C09152=1150.705,51.432,-50.728,-179.726,6.322,149.066
C09153=1150.710,51.184,-50.712,-179.728,6.321,149.066
C09154=1150.715,50.934,-50.696,-179.731,6.319,149.067
C09155=1150.720,50.684,-50.680,-179.733,6.319,149.067
C09156=1150.725,50.435,-50.665,-179.736,6.317,149.068
C09157=1150.730,50.186,-50.650,-179.739,6.317,149.069
C09158=1150.736,49.936,-50.634,-179.741,6.316,149.069
C09159=1150.740,49.686,-50.618,-179.744,6.314,149.069
C09160=1150.745,49.437,-50.603,-179.746,6.314,149.070
C09161=1150.750,49.188,-50.588,-179.749,6.312,149.071
C09162=1150.755,48.938,-50.571,-179.752,6.311,149.071
C09163=1150.760,48.689,-50.555,-179.754,6.310,149.072
C09164=1150.765,48.440,-50.540,-179.757,6.309,149.072
C09165=1150.770,48.190,-50.525,-179.760,6.308,149.073
C09166=1150.775,47.940,-50.509,-179.762,6.307,149.073
C09167=1150.780,47.691,-50.494,-179.765,6.306,149.074
C09168=1150.785,47.442,-50.478,-179.767,6.305,149.074
C09169=1150.791,47.192,-50.463,-179.770,6.304,149.075
C09170=1150.795,46.942,-50.447,-179.773,6.303,149.075
C09171=1150.800,46.693,-50.432,-179.775,6.302,149.076
C09172=1150.805,46.444,-50.416,-179.778,6.301,149.077
C09173=1150.811,46.194,-50.401,-179.780,6.300,149.077
C09174=1150.815,45.945,-50.386,-179.784,6.298,149.078
C09175=1150.820,45.695,-50.370,-179.786,6.298,149.078
C09176=1150.825,45.446,-50.355,-179.789,6.296,149.079
C09177=1150.830,45.197,-50.339,-179.791,6.295,149.079
C09178=1150.836,44.947,-50.324,-179.793,6.295,149.080
C09179=1150.841,44.697,-50.309,-179.797,6.293,149.080
C09180=1150.845,44.447,-50.293,-179.799,6.292,149.081
C09181=1150.851,44.198,-50.278,-179.801,6.291,149.081
C09182=1150.855,43.949,-50.263,-179.804,6.290,149.082
C09183=1150.861,43.699,-50.247,-179.807,6.289,149.082
C09184=1150.865,43.450,-50.232,-179.810,6.288,149.083
C09185=1150.870,43.200,-50.216,-179.812,6.287,149.084
C09186=1150.876,42.951,-50.201,-179.815,6.286,149.084
C09187=1150.881,42.701,-50.186,-179.817,6.285,149.085
C09188=1150.886,42.452,-50.171,-179.820,6.284,149.085
C09189=1150.891,42.203,-50.156,-179.822,6.283,149.086
C09190=1150.896,41.953,-50.140,-179.825,6.282,149.086
C09191=1150.901,41.704,-50.125,-179.828,6.281,149.087
C09192=1150.906,41.453,-50.110,-179.830,6.280,149.087
C09193=1150.910,41.204,-50.095,-179.833,6.279,149.088
C09194=1150.916,40.955,-50.079,-179.835,6.278,149.088
C09195=1150.920,40.706,-50.064,-179.838,6.277,149.089
C09196=1150.926,40.456,-50.049,-179.841,6.276,149.090
C09197=1150.932,40.206,-50.034,-179.843,6.275,149.090
C09198=1150.936,39.957,-50.019,-179.846,6.274,149.091
C09199=1150.942,39.708,-50.003,-179.848,6.273,149.091
C09200=1150.946,39.458,-49.989,-179.851,6.272,149.092
C09201=1150.951,39.208,-49.973,-179.854,6.271,149.092
C09202=1150.956,38.959,-49.958,-179.856,6.270,149.093
C09203=1150.961,38.709,-49.944,-179.859,6.269,149.093
C09204=1150.966,38.460,-49.928,-179.861,6.268,149.094
C09205=1150.971,38.211,-49.913,-179.864,6.267,149.094
C09206=1150.976,37.961,-49.898,-179.867,6.266,149.095
C09207=1150.981,37.712,-49.883,-179.869,6.265,149.095
C09208=1150.987,37.462,-49.868,-179.872,6.264,149.096
C09209=1150.992,37.213,-49.853,-179.874,6.263,149.097
C09210=1150.997,36.963,-49.838,-179.877,6.262,149.097
C09211=1151.002,36.714,-49.823,-179.880,6.261,149.098
C09212=1151.007,36.464,-49.809,-179.882,6.260,149.098
C09213=1151.012,36.215,-49.793,-179.884,6.259,149.099
C09214=1151.017,35.965,-49.779,-179.888,6.258,149.099
C09215=1151.022,35.716,-49.763,-179.890,6.257,149.100
C09216=1151.026,35.466,-49.748,-179.893,6.256,149.100
C09217=1151.031,35.216,-49.734,-179.895,6.255,149.101
C09218=1151.037,34.967,-49.718,-179.897,6.254,149.101
C09219=1151.042,34.717,-49.704,-179.901,6.253,149.102
C09220=1151.047,34.468,-49.688,-179.903,6.252,149.103
C09221=1151.052,34.218,-49.674,-179.906,6.252,149.103
C09222=1151.057,33.969,-49.659,-179.908,6.250,149.104
C09223=1151.062,33.719,-49.644,-179.910,6.249,149.104
C09224=1151.067,33.470,-49.629,-179.913,6.249,149.105
C09225=1151.072,33.220,-49.615,-179.916,6.247,149.105
C09226=1151.077,32.971,-49.599,-179.918,6.247,149.106
C09227=1151.082,32.721,-49.585,-179.921,6.246,149.106
C09228=1151.087,32.472,-49.570,-179.924,6.245,149.107
C09229=1151.093,32.222,-49.555,-179.926,6.244,149.108
C09230=1151.097,31.973,-49.540,-179.929,6.243,149.108
C09231=1151.102,31.723,-49.526,-179.931,6.242,149.109
C09232=1151.108,31.474,-49.512,-179.934,6.241,149.109
C09233=1151.113,31.225,-49.496,-179.937,6.240,149.110
C09234=1151.118,30.975,-49.482,-179.939,6.239,149.110
C09235=1151.123,30.726,-49.467,-179.942,6.238,149.111
C09236=1151.128,30.476,-49.453,-179.944,6.237,149.111
C09237=1151.133,30.226,-49.438,-179.947,6.236,149.112
C09238=1151.138,29.977,-49.423,-179.949,6.235,149.113
C09239=1151.143,29.727,-49.408,-179.952,6.234,149.113
C09240=1151.148,29.478,-49.394,-179.955,6.233,149.114
C09241=1151.153,29.228,-49.379,-179.957,6.232,149.114
C09242=1151.158,28.979,-49.364,-179.959,6.232,149.115
C09243=1151.163,28.729,-49.350,-179.962,6.230,149.115
C09244=1151.168,28.480,-49.335,-179.965,6.230,149.116
C09245=1151.173,28.230,-49.321,-179.967,6.229,149.116
C09246=1151.179,27.961,-49.304,-179.970,6.228,149.117
C09247=1151.185,27.693,-49.289,-179.973,6.227,149.118
C09248=1151.190,27.424,-49.274,-179.976,6.226,149.118
C09249=1151.196,27.154,-49.258,-179.978,6.225,149.119
C09250=1151.201,26.905,-49.244,-179.981,6.224,149.119
C09251=1151.205,26.656,-49.229,-179.984,6.223,149.120
C09252=1151.210,26.406,-49.214,-179.986,6.222,149.120
C09253=1151.215,26.156,-49.200,-179.989,6.221,149.121
C09254=1151.220,25.907,-49.186,-179.991,6.220,149.122
C09255=1151.225,25.657,-49.171,-179.994,6.220,149.122
C09256=1151.231,25.408,-49.156,-179.997,6.218,149.123
C09257=1151.236,25.158,-49.142,-179.999,6.217,149.123
C09258=1151.241,24.909,-49.128,179.998,6.217,149.124
C09259=1151.246,24.659,-49.113,179.996,6.216,149.124
C09260=1151.251,24.409,-49.099,179.993,6.215,149.125
C09261=1151.256,24.160,-49.084,179.991,6.214,149.125
C09262=1151.261,23.911,-49.070,179.988,6.213,149.126
C09263=1151.266,23.661,-49.056,179.985,6.212,149.127
C09264=1151.271,23.412,-49.042,179.983,6.211,149.127
C09265=1151.276,23.162,-49.027,179.981,6.211,149.128
C09266=1151.282,22.912,-49.013,179.978,6.210,149.128
C09267=1151.287,22.662,-48.998,179.975,6.208,149.129
C09268=1151.292,22.413,-48.984,179.973,6.208,149.129
C09269=1151.297,22.164,-48.969,179.970,6.207,149.130
C09270=1151.302,21.914,-48.955,179.968,6.206,149.130
C09271=1151.307,21.665,-48.941,179.965,6.205,149.131
C09272=1151.312,21.415,-48.926,179.963,6.204,149.132
C09273=1151.317,21.166,-48.913,179.960,6.204,149.132
C09274=1151.322,20.916,-48.898,179.957,6.202,149.133
C09275=1151.327,20.667,-48.884,179.955,6.202,149.133
C09276=1151.332,20.417,-48.870,179.953,6.201,149.134
C09277=1151.337,20.167,-48.855,179.949,6.200,149.135
C09278=1151.343,19.918,-48.842,179.947,6.199,149.135
C09279=1151.348,19.668,-48.827,179.945,6.198,149.136
C09280=1151.353,19.419,-48.813,179.942,6.198,149.136
C09281=1151.358,19.169,-48.799,179.940,6.196,149.137
C09282=1151.363,18.920,-48.785,179.937,6.195,149.137
C09283=1151.368,18.670,-48.771,179.935,6.195,149.138
C09284=1151.373,18.421,-48.756,179.932,6.194,149.138
C09285=1151.378,18.171,-48.742,179.929,6.193,149.139
C09286=1151.384,17.922,-48.728,179.927,6.192,149.140
C09287=1151.388,17.673,-48.714,179.925,6.191,149.140
C09288=1151.393,17.422,-48.701,179.922,6.191,149.141
C09289=1151.398,17.172,-48.687,179.919,6.189,149.141
C09290=1151.404,16.923,-48.673,179.917,6.189,149.142
C09291=1151.409,16.674,-48.658,179.914,6.188,149.142
C09292=1151.414,16.424,-48.644,179.912,6.187,149.143
C09293=1151.419,16.175,-48.630,179.909,6.186,149.143
C09294=1151.424,15.925,-48.616,179.906,6.185,149.144
C09295=1151.429,15.676,-48.602,179.904,6.185,149.145
C09296=1151.434,15.425,-48.588,179.902,6.184,149.145
C09297=1151.439,15.177,-48.575,179.899,6.182,149.146
C09298=1151.444,14.927,-48.560,179.897,6.182,149.146
C09299=1151.449,14.677,-48.546,179.894,6.181,149.147
C09300=1151.455,14.428,-48.532,179.892,6.180,149.147
C09301=1151.459,14.178,-48.518,179.889,6.180,149.148
C09302=1151.465,13.928,-48.504,179.886,6.178,149.148
C09303=1151.470,13.679,-48.491,179.884,6.178,149.149
C09304=1151.475,13.430,-48.477,179.881,6.177,149.150
C09305=1151.479,13.180,-48.463,179.879,6.177,149.150
C09306=1151.485,12.930,-48.449,179.876,6.175,149.151
C09307=1151.490,12.681,-48.435,179.873,6.174,149.151
C09308=1151.495,12.431,-48.421,179.871,6.174,149.152
C09309=1151.500,12.182,-48.408,179.869,6.173,149.153
C09310=1151.505,11.932,-48.394,179.866,6.172,149.153
C09311=1151.511,11.683,-48.380,179.864,6.171,149.153
C09312=1151.516,11.433,-48.366,179.861,6.170,149.154
C09313=1151.521,11.183,-48.352,179.859,6.169,149.155
C09314=1151.526,10.934,-48.339,179.856,6.169,149.155
C09315=1151.531,10.684,-48.325,179.854,6.168,149.156
C09316=1151.536,10.434,-48.311,179.851,6.167,149.156
C09317=1151.542,10.185,-48.297,179.849,6.166,149.157
C09318=1151.546,9.936,-48.283,179.846,6.166,149.158
C09319=1151.552,9.686,-48.270,179.844,6.165,149.158
C09320=1151.557,9.436,-48.256,179.841,6.164,149.159
C09321=1151.561,9.187,-48.242,179.838,6.163,149.159
C09322=1151.567,8.937,-48.229,179.836,6.162,149.160
C09323=1151.572,8.688,-48.215,179.834,6.162,149.160
C09324=1151.577,8.439,-48.201,179.831,6.161,149.161
C09325=1151.582,8.189,-48.188,179.829,6.160,149.161
C09326=1151.587,7.940,-48.174,179.825,6.159,149.162
C09327=1151.593,7.689,-48.160,179.823,6.158,149.163
C09328=1151.597,7.440,-48.147,179.821,6.158,149.163
C09329=1151.603,7.190,-48.134,179.818,6.157,149.164
C09330=1151.608,6.941,-48.119,179.816,6.156,149.164
C09331=1151.613,6.691,-48.107,179.813,6.155,149.165
C09332=1151.618,6.442,-48.092,179.811,6.154,149.165
C09333=1151.623,6.193,-48.079,179.808,6.154,149.166
C09334=1151.628,5.942,-48.066,179.806,6.153,149.167
C09335=1151.633,5.693,-48.052,179.803,6.152,149.167
C09336=1151.639,5.443,-48.038,179.801,6.152,149.168
C09337=1151.643,5.194,-48.024,179.798,6.150,149.168
C09338=1151.649,4.944,-48.011,179.796,6.149,149.169
C09339=1151.653,4.694,-47.998,179.793,6.149,149.170
C09340=1151.659,4.445,-47.984,179.791,6.148,149.170
C09341=1151.664,4.195,-47.971,179.788,6.148,149.171
C09342=1151.669,3.946,-47.957,179.786,6.147,149.171
C09343=1151.674,3.696,-47.944,179.783,6.146,149.172
C09344=1151.679,3.447,-47.931,179.781,6.145,149.172
C09345=1151.684,3.197,-47.917,179.778,6.144,149.173
C09346=1151.690,2.947,-47.904,179.776,6.144,149.173
C09347=1151.694,2.698,-47.890,179.773,6.143,149.174
C09348=1151.700,2.448,-47.877,179.771,6.142,149.175
C09349=1151.704,2.199,-47.863,179.768,6.141,149.175
C09350=1151.711,1.929,-47.849,179.766,6.140,149.176
C09351=1151.716,1.660,-47.834,179.763,6.140,149.176
C09352=1151.721,1.390,-47.821,179.760,6.139,149.177
C09353=1151.727,1.121,-47.806,179.758,6.138,149.178
C09354=1151.732,0.871,-47.792,179.755,6.137,149.178
C09355=1151.737,0.622,-47.779,179.753,6.137,149.179
C09356=1151.743,0.372,-47.766,179.750,6.136,149.179
C09357=1151.748,0.123,-47.753,179.748,6.135,149.180
C09358=1151.753,-0.127,-47.739,179.745,6.134,149.181
C09359=1151.758,-0.376,-47.726,179.742,6.133,149.181
C09360=1151.763,-0.627,-47.713,179.740,6.133,149.182
C09361=1151.768,-0.876,-47.700,179.738,6.132,149.182
C09362=1151.774,-1.125,-47.686,179.735,6.132,149.183
C09363=1151.778,-1.375,-47.673,179.733,6.131,149.183
C09364=1151.784,-1.625,-47.660,179.731,6.130,149.184
C09365=1151.789,-1.875,-47.647,179.728,6.130,149.184
C09366=1151.793,-2.123,-47.634,179.725,6.128,149.185
C09367=1151.799,-2.373,-47.620,179.723,6.127,149.186
C09368=1151.804,-2.623,-47.607,179.720,6.127,149.186
C09369=1151.810,-2.873,-47.594,179.718,6.126,149.187
C09370=1151.814,-3.123,-47.581,179.716,6.125,149.187
C09371=1151.820,-3.372,-47.567,179.713,6.125,149.188
C09372=1151.825,-3.621,-47.555,179.711,6.124,149.188
C09373=1151.829,-3.871,-47.542,179.708,6.124,149.189
C09374=1151.835,-4.121,-47.529,179.705,6.122,149.190
C09375=1151.840,-4.371,-47.516,179.703,6.122,149.190
C09376=1151.845,-4.620,-47.502,179.700,6.121,149.191
C09377=1151.850,-4.869,-47.489,179.698,6.120,149.191
C09378=1151.855,-5.119,-47.476,179.696,6.120,149.192
C09379=1151.861,-5.369,-47.463,179.693,6.119,149.193
C09380=1151.866,-5.618,-47.450,179.691,6.118,149.193
C09381=1151.870,-5.868,-47.437,179.688,6.118,149.194
C09382=1151.876,-6.117,-47.424,179.686,6.117,149.194
C09383=1151.881,-6.367,-47.412,179.683,6.116,149.195
C09384=1151.887,-6.617,-47.398,179.680,6.115,149.195
C09385=1151.892,-6.866,-47.385,179.678,6.115,149.196
C09386=1151.897,-7.115,-47.372,179.676,6.114,149.197
C09387=1151.902,-7.365,-47.359,179.673,6.113,149.197
C09388=1151.907,-7.615,-47.346,179.671,6.113,149.198
C09389=1151.912,-7.864,-47.333,179.669,6.112,149.198
C09390=1151.917,-8.114,-47.320,179.666,6.111,149.199
C09391=1151.923,-8.364,-47.307,179.664,6.110,149.199
C09392=1151.928,-8.613,-47.295,179.661,6.110,149.200
C09393=1151.932,-8.863,-47.282,179.659,6.109,149.200
C09394=1151.938,-9.113,-47.268,179.656,6.108,149.201
C09395=1151.943,-9.362,-47.256,179.654,6.107,149.202
C09396=1151.948,-9.612,-47.243,179.651,6.107,149.202
C09397=1151.953,-9.861,-47.230,179.649,6.106,149.203
C09398=1151.959,-10.111,-47.217,179.646,6.106,149.203
C09399=1151.964,-10.360,-47.204,179.644,6.105,149.204
C09400=1151.968,-10.610,-47.192,179.641,6.104,149.205
C09401=1151.973,-10.860,-47.179,179.639,6.103,149.205
C09402=1151.979,-11.109,-47.166,179.636,6.103,149.206
C09403=1151.984,-11.360,-47.153,179.634,6.102,149.206
C09404=1151.989,-11.609,-47.141,179.632,6.102,149.207
C09405=1151.994,-11.859,-47.128,179.629,6.101,149.207
C09406=1152.000,-12.108,-47.116,179.627,6.101,149.208
C09407=1152.005,-12.358,-47.102,179.624,6.099,149.209
C09408=1152.010,-12.608,-47.089,179.621,6.099,149.209
C09409=1152.015,-12.857,-47.077,179.619,6.098,149.210
C09410=1152.020,-13.106,-47.064,179.616,6.097,149.210
C09411=1152.025,-13.356,-47.051,179.614,6.097,149.211
C09412=1152.031,-13.606,-47.039,179.612,6.096,149.211
C09413=1152.036,-13.856,-47.026,179.609,6.095,149.212
C09414=1152.041,-14.105,-47.014,179.607,6.094,149.213
C09415=1152.046,-14.354,-47.001,179.605,6.094,149.213
C09416=1152.051,-14.604,-46.988,179.602,6.093,149.214
C09417=1152.056,-14.854,-46.975,179.600,6.093,149.214
C09418=1152.061,-15.104,-46.964,179.598,6.092,149.215
C09419=1152.067,-15.353,-46.950,179.595,6.092,149.216
C09420=1152.072,-15.603,-46.938,179.593,6.091,149.216
C09421=1152.077,-15.853,-46.925,179.590,6.090,149.217
C09422=1152.082,-16.103,-46.913,179.588,6.090,149.217
C09423=1152.087,-16.352,-46.900,179.585,6.089,149.218
C09424=1152.092,-16.601,-46.888,179.583,6.088,149.218
C09425=1152.098,-16.851,-46.875,179.580,6.088,149.219
C09426=1152.102,-17.101,-46.863,179.578,6.087,149.219
C09427=1152.108,-17.350,-46.850,179.575,6.086,149.220
C09428=1152.113,-17.600,-46.837,179.573,6.085,149.221
C09429=1152.119,-17.849,-46.824,179.570,6.085,149.221
C09430=1152.124,-18.099,-46.813,179.568,6.084,149.222
C09431=1152.129,-18.349,-46.800,179.565,6.083,149.223
C09432=1152.134,-18.598,-46.787,179.563,6.083,149.223
C09433=1152.139,-18.849,-46.775,179.560,6.082,149.224
C09434=1152.144,-19.098,-46.763,179.558,6.081,149.224
C09435=1152.149,-19.347,-46.750,179.556,6.081,149.225
C09436=1152.155,-19.597,-46.738,179.553,6.080,149.225
C09437=1152.160,-19.847,-46.725,179.551,6.079,149.226
C09438=1152.165,-20.096,-46.713,179.549,6.079,149.226
C09439=1152.170,-20.346,-46.701,179.546,6.078,149.227
C09440=1152.176,-20.595,-46.688,179.544,6.078,149.228
C09441=1152.180,-20.845,-46.675,179.542,6.077,149.228
C09442=1152.185,-21.095,-46.664,179.539,6.076,149.229
C09443=1152.191,-21.344,-46.651,179.537,6.076,149.229
C09444=1152.196,-21.594,-46.639,179.534,6.075,149.230
C09445=1152.201,-21.844,-46.626,179.532,6.074,149.230
C09446=1152.207,-22.094,-46.615,179.529,6.074,149.231
C09447=1152.212,-22.343,-46.602,179.527,6.073,149.232
C09448=1152.217,-22.592,-46.589,179.524,6.073,149.232
C09449=1152.222,-22.842,-46.577,179.522,6.072,149.233
C09450=1152.227,-23.091,-46.565,179.520,6.072,149.233
C09451=1152.233,-23.341,-46.553,179.517,6.071,149.234
C09452=1152.237,-23.591,-46.540,179.515,6.070,149.235
C09453=1152.243,-23.841,-46.528,179.512,6.070,149.235
C09454=1152.248,-24.110,-46.515,179.510,6.069,149.236
C09455=1152.254,-24.381,-46.502,179.508,6.068,149.236
C09456=1152.260,-24.651,-46.488,179.505,6.068,149.237
C09457=1152.265,-24.920,-46.475,179.502,6.067,149.238
C09458=1152.271,-25.170,-46.463,179.500,6.066,149.238
C09459=1152.276,-25.420,-46.451,179.497,6.065,149.239
C09460=1152.281,-25.670,-46.439,179.495,6.065,149.239
C09461=1152.286,-25.919,-46.427,179.493,6.065,149.240
C09462=1152.291,-26.169,-46.415,179.490,6.064,149.240
C09463=1152.297,-26.418,-46.403,179.488,6.063,149.241
C09464=1152.302,-26.668,-46.390,179.486,6.063,149.242
C09465=1152.307,-26.918,-46.378,179.483,6.062,149.242
C09466=1152.312,-27.168,-46.365,179.481,6.062,149.243
C09467=1152.317,-27.418,-46.353,179.479,6.061,149.243
C09468=1152.322,-27.668,-46.342,179.476,6.061,149.244
C09469=1152.327,-27.917,-46.330,179.474,6.060,149.244
C09470=1152.332,-28.167,-46.318,179.471,6.059,149.245
C09471=1152.338,-28.417,-46.306,179.469,6.059,149.246
C09472=1152.343,-28.666,-46.293,179.466,6.058,149.246
C09473=1152.348,-28.916,-46.281,179.464,6.057,149.247
C09474=1152.353,-29.165,-46.269,179.461,6.057,149.247
C09475=1152.358,-29.415,-46.257,179.459,6.056,149.248
C09476=1152.364,-29.665,-46.246,179.457,6.056,149.249
C09477=1152.369,-29.913,-46.233,179.454,6.055,149.249
C09478=1152.375,-30.163,-46.221,179.452,6.054,149.250
C09479=1152.379,-30.413,-46.210,179.450,6.054,149.250
C09480=1152.385,-30.663,-46.198,179.447,6.053,149.251
C09481=1152.390,-30.912,-46.186,179.445,6.052,149.251
C09482=1152.395,-31.162,-46.174,179.442,6.052,149.252
C09483=1152.401,-31.412,-46.162,179.440,6.051,149.253
C09484=1152.405,-31.661,-46.150,179.438,6.050,149.253
C09485=1152.411,-31.911,-46.138,179.435,6.050,149.254
C09486=1152.416,-32.161,-46.126,179.433,6.049,149.254
C09487=1152.421,-32.411,-46.114,179.430,6.049,149.255
C09488=1152.426,-32.660,-46.102,179.428,6.048,149.255
C09489=1152.431,-32.910,-46.090,179.425,6.048,149.256
C09490=1152.437,-33.160,-46.078,179.424,6.048,149.257
C09491=1152.442,-33.410,-46.067,179.421,6.047,149.257
C09492=1152.447,-33.659,-46.055,179.419,6.046,149.258
C09493=1152.452,-33.909,-46.043,179.417,6.046,149.258
C09494=1152.457,-34.158,-46.031,179.414,6.045,149.259
C09495=1152.463,-34.407,-46.020,179.412,6.044,149.259
C09496=1152.468,-34.657,-46.008,179.409,6.044,149.260
C09497=1152.474,-34.907,-45.996,179.407,6.043,149.261
C09498=1152.478,-35.156,-45.984,179.404,6.043,149.261
C09499=1152.483,-35.406,-45.972,179.402,6.042,149.262
C09500=1152.489,-35.656,-45.960,179.399,6.042,149.263
C09501=1152.493,-35.906,-45.949,179.397,6.041,149.263
C09502=1152.499,-36.156,-45.937,179.395,6.040,149.264
C09503=1152.504,-36.406,-45.925,179.392,6.040,149.264
C09504=1152.510,-36.655,-45.914,179.390,6.039,149.265
C09505=1152.515,-36.904,-45.902,179.388,6.039,149.265
C09506=1152.520,-37.154,-45.890,179.386,6.038,149.266
C09507=1152.525,-37.403,-45.879,179.383,6.038,149.267
C09508=1152.530,-37.653,-45.867,179.381,6.037,149.267
C09509=1152.536,-37.903,-45.855,179.378,6.037,149.268
C09510=1152.540,-38.153,-45.844,179.376,6.036,149.268
C09511=1152.546,-38.402,-45.832,179.374,6.036,149.269
C09512=1152.552,-38.652,-45.820,179.371,6.035,149.269
C09513=1152.557,-38.902,-45.809,179.369,6.034,149.270
C09514=1152.562,-39.152,-45.797,179.367,6.034,149.271
C09515=1152.567,-39.401,-45.786,179.364,6.033,149.271
C09516=1152.572,-39.651,-45.774,179.362,6.032,149.272
C09517=1152.578,-39.900,-45.762,179.360,6.032,149.272
C09518=1152.583,-40.150,-45.751,179.357,6.032,149.273
C09519=1152.588,-40.400,-45.739,179.355,6.031,149.273
C09520=1152.593,-40.650,-45.728,179.353,6.031,149.274
C09521=1152.598,-40.900,-45.716,179.350,6.030,149.275
C09522=1152.604,-41.149,-45.705,179.348,6.030,149.275
C09523=1152.609,-41.398,-45.693,179.346,6.029,149.276
C09524=1152.614,-41.648,-45.682,179.343,6.028,149.276
C09525=1152.619,-41.898,-45.670,179.341,6.028,149.277
C09526=1152.624,-42.148,-45.659,179.339,6.027,149.277
C09527=1152.630,-42.397,-45.647,179.337,6.027,149.278
C09528=1152.635,-42.647,-45.635,179.334,6.026,149.279
C09529=1152.640,-42.896,-45.624,179.332,6.026,149.279
C09530=1152.646,-43.147,-45.613,179.329,6.025,149.280
C09531=1152.650,-43.397,-45.601,179.327,6.025,149.280
C09532=1152.657,-43.646,-45.590,179.325,6.024,149.281
C09533=1152.661,-43.895,-45.579,179.322,6.024,149.282
C09534=1152.667,-44.145,-45.567,179.320,6.023,149.282
C09535=1152.671,-44.395,-45.555,179.317,6.022,149.283
C09536=1152.677,-44.644,-45.545,179.316,6.022,149.283
C09537=1152.682,-44.894,-45.533,179.313,6.022,149.284
C09538=1152.687,-45.144,-45.522,179.311,6.021,149.284
C09539=1152.692,-45.394,-45.510,179.308,6.020,149.285
C09540=1152.698,-45.643,-45.499,179.306,6.020,149.286
C09541=1152.703,-45.893,-45.487,179.304,6.019,149.286
C09542=1152.708,-46.143,-45.476,179.301,6.019,149.287
C09543=1152.713,-46.393,-45.464,179.299,6.018,149.287
C09544=1152.719,-46.642,-45.454,179.297,6.018,149.288
C09545=1152.724,-46.892,-45.442,179.295,6.018,149.288
C09546=1152.729,-47.142,-45.431,179.292,6.017,149.289
C09547=1152.734,-47.391,-45.420,179.290,6.016,149.290
C09548=1152.740,-47.640,-45.408,179.287,6.016,149.290
C09549=1152.745,-47.891,-45.397,179.285,6.015,149.291
C09550=1152.750,-48.141,-45.386,179.283,6.014,149.291
C09551=1152.755,-48.390,-45.375,179.281,6.015,149.292
C09552=1152.760,-48.639,-45.363,179.278,6.014,149.292
C09553=1152.766,-48.890,-45.352,179.276,6.013,149.293
C09554=1152.771,-49.139,-45.341,179.274,6.013,149.294
C09555=1152.777,-49.389,-45.329,179.271,6.012,149.294
C09556=1152.782,-49.639,-45.319,179.269,6.012,149.295
C09557=1152.787,-49.888,-45.308,179.266,6.011,149.295
C09558=1152.793,-50.159,-45.296,179.264,6.010,149.296
C09559=1152.798,-50.430,-45.283,179.262,6.010,149.296
C09560=1152.804,-50.700,-45.271,179.259,6.009,149.297
C09561=1152.810,-50.970,-45.259,179.256,6.009,149.298
C09562=1152.815,-51.220,-45.248,179.255,6.009,149.298
C09563=1152.820,-51.470,-45.237,179.252,6.008,149.299
C09564=1152.825,-51.719,-45.225,179.250,6.008,149.300
C09565=1152.831,-51.969,-45.215,179.248,6.007,149.300
C09566=1152.836,-52.219,-45.204,179.245,6.006,149.301
C09567=1152.841,-52.469,-45.193,179.243,6.006,149.301
C09568=1152.847,-52.718,-45.182,179.240,6.005,149.302
C09569=1152.851,-52.968,-45.170,179.239,6.005,149.302
C09570=1152.856,-53.218,-45.160,179.236,6.005,149.303
C09571=1152.862,-53.467,-45.148,179.234,6.004,149.304
C09572=1152.867,-53.717,-45.138,179.231,6.003,149.304
C09573=1152.872,-53.967,-45.126,179.229,6.003,149.305
C09574=1152.877,-54.216,-45.115,179.227,6.002,149.305
C09575=1152.883,-54.467,-45.104,179.225,6.003,149.306
C09576=1152.888,-54.716,-45.093,179.222,6.002,149.306
C09577=1152.893,-54.966,-45.083,179.220,6.001,149.307
C09578=1152.898,-55.215,-45.071,179.218,6.001,149.308
C09579=1152.904,-55.465,-45.061,179.215,6.000,149.308
C09580=1152.909,-55.715,-45.049,179.213,6.000,149.309
C09581=1152.915,-55.964,-45.039,179.211,5.999,149.309
C09582=1152.919,-56.214,-45.028,179.208,5.999,149.310
C09583=1152.924,-56.464,-45.017,179.206,5.998,149.310
C09584=1152.930,-56.714,-45.006,179.204,5.998,149.311
C09585=1152.935,-56.964,-44.995,179.201,5.997,149.312
C09586=1152.941,-57.213,-44.984,179.200,5.997,149.312
C09587=1152.946,-57.463,-44.974,179.197,5.997,149.313
C09588=1152.951,-57.712,-44.963,179.195,5.996,149.313
C09589=1152.957,-57.962,-44.952,179.192,5.995,149.314
C09590=1152.962,-58.212,-44.940,179.190,5.995,149.314
C09591=1152.967,-58.462,-44.930,179.188,5.995,149.315
C09592=1152.972,-58.711,-44.919,179.186,5.994,149.316
C09593=1152.977,-58.961,-44.909,179.184,5.994,149.316
C09594=1152.982,-59.210,-44.897,179.181,5.993,149.317
C09595=1152.988,-59.460,-44.886,179.179,5.992,149.317
C09596=1152.993,-59.710,-44.876,179.177,5.992,149.318
C09597=1152.999,-59.959,-44.865,179.174,5.992,149.318
C09598=1153.004,-60.210,-44.854,179.172,5.991,149.319
C09599=1153.008,-60.459,-44.843,179.170,5.991,149.320
C09600=1153.014,-60.709,-44.833,179.167,5.990,149.320
C09601=1153.019,-60.959,-44.822,179.165,5.990,149.321
C09602=1153.024,-61.208,-44.811,179.163,5.990,149.321
C09603=1153.030,-61.459,-44.800,179.161,5.989,149.322
C09604=1153.035,-61.707,-44.789,179.158,5.988,149.322
C09605=1153.040,-61.958,-44.779,179.156,5.988,149.323
C09606=1153.046,-62.207,-44.769,179.154,5.988,149.324
C09607=1153.051,-62.457,-44.757,179.152,5.987,149.324
C09608=1153.056,-62.706,-44.747,179.150,5.987,149.325
C09609=1153.061,-62.957,-44.736,179.147,5.986,149.325
C09610=1153.067,-63.206,-44.726,179.145,5.985,149.326
C09611=1153.071,-63.456,-44.715,179.143,5.986,149.327
C09612=1153.077,-63.705,-44.705,179.141,5.985,149.327
C09613=1153.082,-63.956,-44.694,179.138,5.984,149.327
C09614=1153.087,-64.205,-44.683,179.136,5.984,149.328
C09615=1153.093,-64.455,-44.672,179.134,5.984,149.329
C09616=1153.099,-64.705,-44.662,179.131,5.983,149.329
C09617=1153.104,-64.954,-44.652,179.129,5.983,149.330
C09618=1153.109,-65.204,-44.640,179.127,5.982,149.330
C09619=1153.115,-65.453,-44.630,179.124,5.981,149.331
C09620=1153.120,-65.704,-44.620,179.123,5.981,149.332
C09621=1153.125,-65.953,-44.609,179.120,5.981,149.332
C09622=1153.130,-66.203,-44.598,179.118,5.980,149.333
C09623=1153.135,-66.452,-44.588,179.116,5.980,149.333
C09624=1153.140,-66.703,-44.577,179.114,5.980,149.334
C09625=1153.146,-66.952,-44.567,179.111,5.979,149.334
C09626=1153.152,-67.202,-44.557,179.109,5.979,149.335
C09627=1153.156,-67.451,-44.546,179.107,5.978,149.336
C09628=1153.162,-67.701,-44.535,179.105,5.978,149.336
C09629=1153.167,-67.951,-44.525,179.102,5.978,149.337
C09630=1153.173,-68.201,-44.515,179.100,5.977,149.337
C09631=1153.178,-68.451,-44.504,179.098,5.976,149.338
C09632=1153.183,-68.700,-44.494,179.096,5.976,149.338
C09633=1153.188,-68.949,-44.483,179.094,5.976,149.339
C09634=1153.193,-69.200,-44.472,179.091,5.975,149.340
C09635=1153.198,-69.449,-44.463,179.089,5.975,149.340
C09636=1153.203,-69.699,-44.452,179.087,5.974,149.341
C09637=1153.209,-69.949,-44.442,179.085,5.974,149.341
C09638=1153.215,-70.198,-44.432,179.082,5.973,149.342
C09639=1153.220,-70.448,-44.421,179.080,5.973,149.342
C09640=1153.225,-70.698,-44.411,179.078,5.973,149.343
C09641=1153.230,-70.947,-44.400,179.076,5.972,149.343
C09642=1153.235,-71.197,-44.389,179.073,5.972,149.344
C09643=1153.241,-71.447,-44.379,179.071,5.971,149.345
C09644=1153.246,-71.697,-44.369,179.070,5.971,149.345
C09645=1153.252,-71.946,-44.358,179.067,5.971,149.346
C09646=1153.257,-72.196,-44.348,179.065,5.970,149.346
C09647=1153.262,-72.446,-44.338,179.062,5.970,149.347
C09648=1153.267,-72.695,-44.328,179.060,5.970,149.347
C09649=1153.273,-72.945,-44.318,179.058,5.969,149.348
C09650=1153.278,-73.195,-44.307,179.056,5.968,149.349
C09651=1153.283,-73.445,-44.297,179.053,5.968,149.349
C09652=1153.289,-73.694,-44.287,179.052,5.968,149.350
C09653=1153.294,-73.945,-44.276,179.049,5.967,149.350
C09654=1153.299,-74.194,-44.266,179.047,5.966,149.351
C09655=1153.304,-74.443,-44.256,179.044,5.966,149.352
C09656=1153.309,-74.694,-44.246,179.043,5.966,149.352
C09657=1153.315,-74.943,-44.236,179.040,5.965,149.352
C09658=1153.320,-75.193,-44.225,179.038,5.965,149.353
C09659=1153.325,-75.443,-44.215,179.036,5.965,149.354
C09660=1153.331,-75.692,-44.205,179.034,5.964,149.354
C09661=1153.337,-75.942,-44.194,179.031,5.964,149.355
C09662=1153.342,-76.213,-44.184,179.029,5.963,149.355
C09663=1153.347,-76.485,-44.173,179.026,5.963,149.356
C09664=1153.354,-76.756,-44.162,179.025,5.963,149.357
C09665=1153.359,-77.027,-44.151,179.022,5.962,149.357
C09666=1153.365,-77.277,-44.141,179.020,5.962,149.358
C09667=1153.370,-77.527,-44.130,179.017,5.961,149.358
C09668=1153.375,-77.777,-44.120,179.016,5.961,149.359
C09669=1153.381,-78.026,-44.110,179.013,5.960,149.359
C09670=1153.386,-78.275,-44.100,179.011,5.960,149.360
C09671=1153.391,-78.526,-44.090,179.009,5.959,149.361
C09672=1153.397,-78.776,-44.080,179.007,5.959,149.361
C09673=1153.402,-79.025,-44.070,179.004,5.959,149.362
C09674=1153.407,-79.275,-44.060,179.002,5.958,149.362
C09675=1153.412,-79.525,-44.050,179.000,5.959,149.363
C09676=1153.418,-79.774,-44.040,178.998,5.958,149.363
C09677=1153.423,-80.024,-44.029,178.996,5.957,149.364
C09678=1153.428,-80.274,-44.021,178.993,5.957,149.365
C09679=1153.433,-80.524,-44.010,178.991,5.957,149.365
C09680=1153.439,-80.774,-44.000,178.989,5.956,149.366
C09681=1153.445,-81.023,-43.990,178.987,5.955,149.366
C09682=1153.450,-81.272,-43.980,178.985,5.955,149.367
C09683=1153.455,-81.523,-43.970,178.983,5.955,149.367
C09684=1153.460,-81.773,-43.960,178.980,5.954,149.368
C09685=1153.465,-82.022,-43.950,178.979,5.954,149.368
C09686=1153.471,-82.272,-43.940,178.976,5.954,149.369
C09687=1153.476,-82.521,-43.930,178.974,5.953,149.370
C09688=1153.481,-82.772,-43.921,178.972,5.953,149.370
C09689=1153.487,-83.021,-43.910,178.970,5.952,149.371
C09690=1153.492,-83.271,-43.900,178.967,5.952,149.371
C09691=1153.497,-83.520,-43.891,178.965,5.951,149.372
C09692=1153.502,-83.771,-43.881,178.963,5.951,149.372
C09693=1153.508,-84.020,-43.871,178.961,5.951,149.373
C09694=1153.513,-84.270,-43.861,178.959,5.950,149.374
C09695=1153.519,-84.520,-43.851,178.957,5.950,149.374
C09696=1153.524,-84.769,-43.841,178.954,5.950,149.375
C09697=1153.529,-85.019,-43.831,178.952,5.949,149.375
C09698=1153.535,-85.269,-43.822,178.950,5.949,149.376
C09699=1153.539,-85.519,-43.812,178.948,5.949,149.376
C09700=1153.545,-85.768,-43.802,178.946,5.948,149.377
C09701=1153.551,-86.018,-43.792,178.944,5.948,149.377
C09702=1153.556,-86.268,-43.783,178.941,5.948,149.378
C09703=1153.561,-86.518,-43.772,178.939,5.947,149.379
C09704=1153.566,-86.768,-43.763,178.938,5.947,149.379
C09705=1153.572,-87.017,-43.753,178.935,5.946,149.380
C09706=1153.577,-87.267,-43.743,178.933,5.946,149.380
C09707=1153.582,-87.517,-43.734,178.931,5.946,149.381
C09708=1153.588,-87.766,-43.724,178.928,5.945,149.381
C09709=1153.592,-88.016,-43.714,178.926,5.945,149.382
C09710=1153.598,-88.266,-43.704,178.925,5.945,149.382
C09711=1153.603,-88.516,-43.695,178.922,5.944,149.383
C09712=1153.609,-88.766,-43.685,178.920,5.943,149.384
C09713=1153.614,-89.015,-43.675,178.918,5.943,149.384
C09714=1153.619,-89.264,-43.665,178.916,5.943,149.385
C09715=1153.625,-89.515,-43.656,178.913,5.942,149.385
C09716=1153.630,-89.764,-43.646,178.912,5.942,149.386
C09717=1153.635,-90.015,-43.636,178.910,5.942,149.386
C09718=1153.640,-90.264,-43.627,178.907,5.941,149.387
C09719=1153.646,-90.514,-43.617,178.905,5.941,149.387
C09720=1153.651,-90.763,-43.608,178.903,5.940,149.388
C09721=1153.657,-91.014,-43.598,178.900,5.940,149.389
C09722=1153.662,-91.263,-43.589,178.899,5.940,149.389
C09723=1153.668,-91.513,-43.579,178.897,5.939,149.390
C09724=1153.672,-91.762,-43.570,178.895,5.940,149.390
C09725=1153.678,-92.012,-43.560,178.892,5.939,149.391
C09726=1153.683,-92.262,-43.550,178.890,5.938,149.391
C09727=1153.689,-92.512,-43.541,178.888,5.939,149.392
C09728=1153.693,-92.762,-43.531,178.886,5.938,149.392
C09729=1153.699,-93.012,-43.521,178.884,5.937,149.393
C09730=1153.704,-93.261,-43.512,178.882,5.937,149.393
C09731=1153.710,-93.511,-43.502,178.879,5.937,149.394
C09732=1153.715,-93.760,-43.493,178.877,5.936,149.395
C09733=1153.721,-94.011,-43.483,178.876,5.936,149.395
C09734=1153.726,-94.260,-43.474,178.873,5.936,149.396
C09735=1153.731,-94.510,-43.465,178.871,5.936,149.396
C09736=1153.737,-94.760,-43.455,178.869,5.935,149.397
C09737=1153.742,-95.009,-43.446,178.866,5.935,149.398
C09738=1153.748,-95.259,-43.436,178.865,5.935,149.398
C09739=1153.752,-95.508,-43.427,178.863,5.934,149.398
C09740=1153.758,-95.759,-43.417,178.860,5.933,149.399
C09741=1153.763,-96.008,-43.407,178.858,5.933,149.400
C09742=1153.768,-96.258,-43.399,178.856,5.933,149.400
C09743=1153.774,-96.508,-43.389,178.854,5.932,149.401
C09744=1153.778,-96.758,-43.379,178.852,5.932,149.401
C09745=1153.784,-97.008,-43.370,178.850,5.932,149.402
C09746=1153.790,-97.258,-43.361,178.848,5.932,149.402
C09747=1153.794,-97.507,-43.351,178.846,5.931,149.403
C09748=1153.800,-97.757,-43.342,178.843,5.931,149.404
C09749=1153.805,-98.007,-43.333,178.842,5.931,149.404
C09750=1153.811,-98.257,-43.322,178.840,5.930,149.404
C09751=1153.816,-98.506,-43.314,178.838,5.930,149.405
C09752=1153.821,-98.756,-43.305,178.835,5.929,149.406
C09753=1153.827,-99.006,-43.294,178.833,5.929,149.406
C09754=1153.832,-99.256,-43.286,178.831,5.929,149.407
C09755=1153.837,-99.506,-43.277,178.829,5.928,149.407
C09756=1153.843,-99.755,-43.266,178.827,5.928,149.408
C09757=1153.848,-100.005,-43.258,178.825,5.928,149.408
C09758=1153.854,-100.255,-43.248,178.823,5.927,149.409
C09759=1153.860,-100.504,-43.239,178.821,5.927,149.410
C09760=1153.865,-100.753,-43.230,178.819,5.926,149.410
C09761=1153.870,-101.003,-43.221,178.816,5.926,149.411
C09762=1153.876,-101.254,-43.211,178.815,5.926,149.411
C09763=1153.881,-101.503,-43.203,178.812,5.925,149.412
C09764=1153.886,-101.753,-43.193,178.810,5.925,149.412
C09765=1153.892,-102.003,-43.183,178.808,5.925,149.413
C09766=1153.897,-102.275,-43.173,178.806,5.924,149.413
C09767=1153.903,-102.547,-43.164,178.804,5.924,149.414
C09768=1153.908,-102.819,-43.154,178.801,5.924,149.415
C09769=1153.914,-103.091,-43.143,178.799,5.923,149.415
C09770=1153.920,-103.341,-43.134,178.797,5.922,149.416
C09771=1153.925,-103.591,-43.125,178.795,5.923,149.416
C09772=1153.931,-103.840,-43.116,178.793,5.922,149.417
C09773=1153.936,-104.090,-43.107,178.791,5.922,149.417
C09774=1153.942,-104.340,-43.097,178.789,5.921,149.418
C09775=1153.947,-104.589,-43.088,178.786,5.921,149.418
C09776=1153.952,-104.839,-43.079,178.785,5.921,149.419
C09777=1153.957,-105.089,-43.071,178.782,5.920,149.419
C09778=1153.963,-105.339,-43.061,178.781,5.920,149.420
C09779=1153.968,-105.589,-43.052,178.778,5.920,149.421
C09780=1153.973,-105.838,-43.043,178.777,5.920,149.421
C09781=1153.978,-106.088,-43.034,178.774,5.919,149.422
C09782=1153.983,-106.338,-43.025,178.772,5.918,149.422
C09783=1153.989,-106.588,-43.015,178.770,5.919,149.423
C09784=1153.994,-106.838,-43.006,178.768,5.918,149.423
C09785=1154.000,-107.087,-42.998,178.766,5.918,149.424
C09786=1154.005,-107.337,-42.989,178.764,5.917,149.424
C09787=1154.010,-107.587,-42.980,178.762,5.917,149.425
C09788=1154.016,-107.837,-42.971,178.760,5.917,149.425
C09789=1154.022,-108.087,-42.962,178.758,5.916,149.426
C09790=1154.026,-108.336,-42.952,178.756,5.916,149.426
C09791=1154.032,-108.586,-42.943,178.754,5.916,149.427
C09792=1154.037,-108.836,-42.934,178.752,5.916,149.428
C09793=1154.042,-109.085,-42.926,178.750,5.915,149.428
C09794=1154.048,-109.335,-42.916,178.748,5.915,149.429
C09795=1154.054,-109.585,-42.907,178.746,5.915,149.429
C09796=1154.059,-109.835,-42.898,178.743,5.914,149.430
C09797=1154.064,-110.085,-42.890,178.741,5.914,149.430
C09798=1154.069,-110.335,-42.881,178.739,5.913,149.431
C09799=1154.074,-110.585,-42.872,178.738,5.913,149.431
C09800=1154.080,-110.834,-42.863,178.735,5.913,149.432
C09801=1154.086,-111.084,-42.854,178.733,5.913,149.432
C09802=1154.091,-111.334,-42.845,178.731,5.912,149.433
C09803=1154.096,-111.584,-42.836,178.729,5.912,149.433
C09804=1154.101,-111.833,-42.827,178.727,5.912,149.434
C09805=1154.107,-112.083,-42.818,178.725,5.911,149.435
C09806=1154.112,-112.332,-42.810,178.723,5.911,149.435
C09807=1154.118,-112.582,-42.801,178.721,5.911,149.436
C09808=1154.123,-112.832,-42.792,178.719,5.911,149.436
C09809=1154.129,-113.082,-42.782,178.717,5.910,149.437
C09810=1154.134,-113.332,-42.773,178.715,5.910,149.437
C09811=1154.139,-113.582,-42.765,178.713,5.910,149.438
C09812=1154.145,-113.832,-42.757,178.711,5.909,149.438
C09813=1154.150,-114.082,-42.748,178.709,5.909,149.439
C09814=1154.155,-114.331,-42.739,178.707,5.908,149.439
C09815=1154.160,-114.581,-42.730,178.705,5.908,149.440
C09816=1154.166,-114.831,-42.721,178.703,5.908,149.440
C09817=1154.171,-115.080,-42.713,178.701,5.908,149.441
C09818=1154.177,-115.330,-42.704,178.699,5.907,149.441
C09819=1154.182,-115.580,-42.695,178.697,5.907,149.442
C09820=1154.187,-115.830,-42.686,178.695,5.907,149.443
C09821=1154.193,-116.079,-42.677,178.693,5.907,149.443
C09822=1154.198,-116.329,-42.669,178.691,5.906,149.444
C09823=1154.203,-116.579,-42.660,178.689,5.905,149.444
C09824=1154.208,-116.829,-42.651,178.687,5.905,149.445
C09825=1154.214,-117.079,-42.642,178.685,5.904,149.445
C09826=1154.219,-117.328,-42.634,178.683,5.905,149.446
C09827=1154.225,-117.578,-42.625,178.680,5.904,149.446
C09828=1154.230,-117.828,-42.617,178.679,5.904,149.447
C09829=1154.235,-118.078,-42.608,178.677,5.903,149.447
C09830=1154.241,-118.327,-42.599,178.675,5.903,149.448
C09831=1154.246,-118.577,-42.591,178.672,5.903,149.448
C09832=1154.251,-118.827,-42.582,178.671,5.903,149.449
C09833=1154.257,-119.078,-42.573,178.669,5.902,149.449
C09834=1154.263,-119.327,-42.565,178.667,5.902,149.450
C09835=1154.268,-119.577,-42.556,178.665,5.902,149.450
C09836=1154.273,-119.826,-42.547,178.663,5.902,149.451
C09837=1154.278,-120.076,-42.538,178.661,5.901,149.452
C09838=1154.284,-120.326,-42.530,178.658,5.901,149.452
C09839=1154.289,-120.576,-42.522,178.657,5.901,149.453
C09840=1154.294,-120.826,-42.513,178.655,5.900,149.453
C09841=1154.300,-121.075,-42.504,178.653,5.900,149.454
C09842=1154.306,-121.325,-42.496,178.651,5.899,149.454
C09843=1154.311,-121.575,-42.487,178.649,5.900,149.455
C09844=1154.316,-121.825,-42.478,178.646,5.899,149.455
C09845=1154.322,-122.074,-42.470,178.645,5.899,149.456
C09846=1154.327,-122.325,-42.461,178.643,5.898,149.456
C09847=1154.332,-122.575,-42.452,178.641,5.898,149.457
C09848=1154.338,-122.824,-42.444,178.639,5.897,149.457
C09849=1154.343,-123.074,-42.436,178.637,5.898,149.458
C09850=1154.348,-123.324,-42.427,178.635,5.897,149.458
C09851=1154.354,-123.573,-42.419,178.633,5.897,149.459
C09852=1154.359,-123.823,-42.411,178.631,5.896,149.459
C09853=1154.365,-124.073,-42.402,178.629,5.896,149.460
C09854=1154.370,-124.322,-42.393,178.627,5.896,149.460
C09855=1154.376,-124.573,-42.385,178.625,5.896,149.461
C09856=1154.381,-124.823,-42.376,178.623,5.895,149.462
C09857=1154.387,-125.072,-42.368,178.621,5.895,149.462
C09858=1154.391,-125.322,-42.360,178.619,5.895,149.462
C09859=1154.397,-125.572,-42.351,178.617,5.895,149.463
C09860=1154.402,-125.821,-42.343,178.615,5.894,149.463
C09861=1154.408,-126.071,-42.335,178.614,5.894,149.464
C09862=1154.413,-126.321,-42.326,178.611,5.893,149.464
C09863=1154.419,-126.571,-42.318,178.609,5.894,149.465
C09864=1154.424,-126.821,-42.309,178.607,5.893,149.466
C09865=1154.429,-127.071,-42.301,178.606,5.893,149.466
C09866=1154.435,-127.320,-42.293,178.603,5.892,149.467
C09867=1154.440,-127.570,-42.284,178.602,5.892,149.467
C09868=1154.445,-127.821,-42.276,178.600,5.891,149.468
C09869=1154.451,-128.070,-42.267,178.598,5.892,149.468
C09870=1154.030,-128.081,-42.310,178.594,5.895,149.470
C09871=1154.024,-127.831,-42.318,178.596,5.896,149.469
C09872=1154.019,-127.582,-42.326,178.598,5.895,149.469
C09873=1154.014,-127.332,-42.335,178.600,5.896,149.468
C09874=1154.008,-127.081,-42.343,178.602,5.896,149.468
C09875=1154.003,-126.832,-42.351,178.604,5.897,149.467
C09876=1153.998,-126.582,-42.360,178.606,5.897,149.467
C09877=1153.992,-126.332,-42.368,178.608,5.897,149.466
C09878=1153.987,-126.083,-42.377,178.610,5.897,149.466
C09879=1153.981,-125.833,-42.385,178.612,5.898,149.465
C09880=1153.976,-125.583,-42.394,178.614,5.898,149.465
C09881=1153.971,-125.333,-42.401,178.616,5.899,149.464
C09882=1153.965,-125.083,-42.410,178.617,5.899,149.464
C09883=1153.960,-124.834,-42.419,178.620,5.899,149.463
C09884=1153.954,-124.584,-42.427,178.622,5.899,149.463
C09885=1153.949,-124.334,-42.436,178.624,5.900,149.462
C09886=1153.944,-124.084,-42.445,178.625,5.900,149.462
C09887=1153.938,-123.834,-42.452,178.628,5.900,149.461
C09888=1153.933,-123.584,-42.461,178.629,5.900,149.461
C09889=1153.928,-123.335,-42.470,178.631,5.901,149.460
C09890=1153.922,-123.085,-42.478,178.633,5.901,149.459
C09891=1153.917,-122.835,-42.486,178.636,5.901,149.459
C09892=1153.912,-122.585,-42.495,178.637,5.901,149.458
C09893=1153.906,-122.336,-42.503,178.639,5.902,149.458
C09894=1153.901,-122.086,-42.512,178.641,5.902,149.458
C09895=1153.895,-121.836,-42.521,178.643,5.903,149.457
C09896=1153.890,-121.587,-42.529,178.645,5.903,149.457
C09897=1153.884,-121.336,-42.538,178.648,5.903,149.456
C09898=1153.879,-121.086,-42.547,178.649,5.903,149.455
C09899=1153.874,-120.837,-42.555,178.651,5.904,149.455
C09900=1153.868,-120.587,-42.564,178.653,5.904,149.454
C09901=1153.863,-120.337,-42.572,178.655,5.905,149.454
C09902=1153.857,-120.087,-42.581,178.657,5.905,149.453
C09903=1153.853,-119.838,-42.589,178.659,5.905,149.453
C09904=1153.847,-119.588,-42.598,178.661,5.905,149.452
C09905=1153.842,-119.338,-42.606,178.663,5.906,149.452
C09906=1153.837,-119.088,-42.615,178.665,5.906,149.451
C09907=1153.831,-118.839,-42.623,178.667,5.906,149.451
C09908=1153.826,-118.589,-42.632,178.669,5.907,149.450
C09909=1153.820,-118.339,-42.641,178.671,5.907,149.450
C09910=1153.815,-118.089,-42.649,178.673,5.907,149.449
C09911=1153.809,-117.840,-42.658,178.675,5.907,149.449
C09912=1153.804,-117.590,-42.667,178.677,5.908,149.448
C09913=1153.799,-117.340,-42.676,178.679,5.908,149.448
C09914=1153.794,-117.090,-42.685,178.682,5.909,149.447
C09915=1153.788,-116.840,-42.693,178.683,5.908,149.446
C09916=1153.783,-116.590,-42.701,178.685,5.909,149.446
C09917=1153.777,-116.341,-42.710,178.687,5.909,149.445
C09918=1153.772,-116.091,-42.719,178.689,5.910,149.445
C09919=1153.767,-115.841,-42.728,178.691,5.910,149.444
C09920=1153.761,-115.591,-42.737,178.693,5.910,149.444
C09921=1153.755,-115.342,-42.746,178.696,5.911,149.443
C09922=1153.750,-115.092,-42.755,178.697,5.911,149.443
C09923=1153.745,-114.841,-42.763,178.699,5.912,149.442
C09924=1153.739,-114.592,-42.772,178.701,5.912,149.442
C09925=1153.734,-114.342,-42.781,178.704,5.912,149.441
C09926=1153.729,-114.092,-42.790,178.705,5.912,149.441
C09927=1153.723,-113.843,-42.798,178.707,5.913,149.440
C09928=1153.718,-113.593,-42.807,178.709,5.913,149.440
C09929=1153.713,-113.344,-42.816,178.711,5.914,149.439
C09930=1153.707,-113.094,-42.825,178.713,5.913,149.438
C09931=1153.702,-112.844,-42.834,178.715,5.914,149.438
C09932=1153.697,-112.594,-42.843,178.718,5.915,149.437
C09933=1153.691,-112.344,-42.852,178.719,5.915,149.437
C09934=1153.686,-112.094,-42.861,178.721,5.915,149.436
C09935=1153.680,-111.845,-42.869,178.724,5.915,149.436
C09936=1153.675,-111.595,-42.878,178.726,5.916,149.435
C09937=1153.670,-111.345,-42.887,178.727,5.916,149.435
C09938=1153.665,-111.095,-42.896,178.730,5.916,149.434
C09939=1153.660,-110.845,-42.905,178.732,5.917,149.434
C09940=1153.654,-110.596,-42.914,178.734,5.917,149.433
C09941=1153.649,-110.346,-42.922,178.736,5.917,149.433
C09942=1153.643,-110.096,-42.932,178.738,5.917,149.432
C09943=1153.637,-109.846,-42.941,178.740,5.918,149.432
C09944=1153.632,-109.597,-42.950,178.742,5.918,149.431
C09945=1153.627,-109.347,-42.959,178.744,5.919,149.430
C09946=1153.622,-109.097,-42.968,178.746,5.918,149.430
C09947=1153.617,-108.847,-42.976,178.748,5.919,149.429
C09948=1153.610,-108.598,-42.986,178.750,5.920,149.429
C09949=1153.605,-108.348,-42.995,178.752,5.920,149.428
C09950=1153.600,-108.098,-43.003,178.754,5.920,149.428
C09951=1153.595,-107.848,-43.012,178.756,5.920,149.427
C09952=1153.590,-107.598,-43.021,178.758,5.921,149.427
C09953=1153.584,-107.348,-43.030,178.761,5.921,149.426
C09954=1153.579,-107.098,-43.040,178.762,5.921,149.426
C09955=1153.573,-106.848,-43.048,178.765,5.922,149.425
C09956=1153.568,-106.598,-43.057,178.766,5.922,149.425
C09957=1153.563,-106.350,-43.067,178.769,5.922,149.424
C09958=1153.558,-106.100,-43.076,178.770,5.922,149.423
C09959=1153.552,-105.850,-43.085,178.773,5.923,149.423
C09960=1153.547,-105.600,-43.094,178.775,5.924,149.422
C09961=1153.541,-105.350,-43.103,178.776,5.924,149.422
C09962=1153.536,-105.100,-43.112,178.779,5.924,149.421
C09963=1153.530,-104.850,-43.121,178.781,5.924,149.421
C09964=1153.525,-104.600,-43.130,178.783,5.925,149.420
C09965=1153.520,-104.351,-43.140,178.785,5.926,149.420
C09966=1153.515,-104.101,-43.149,178.787,5.925,149.419
C09967=1153.509,-103.851,-43.158,178.789,5.926,149.419
C09968=1153.504,-103.601,-43.167,178.791,5.926,149.418
C09969=1153.499,-103.351,-43.176,178.793,5.927,149.418
C09970=1153.493,-103.103,-43.185,178.795,5.926,149.417
C09971=1153.487,-102.830,-43.195,178.797,5.927,149.416
C09972=1153.481,-102.558,-43.205,178.800,5.928,149.416
C09973=1153.476,-102.286,-43.216,178.802,5.928,149.415
C09974=1153.470,-102.014,-43.225,178.804,5.928,149.415
C09975=1153.465,-101.764,-43.235,178.807,5.929,149.414
C09976=1153.459,-101.514,-43.244,178.809,5.929,149.414
C09977=1153.454,-101.264,-43.253,178.810,5.929,149.413
C09978=1153.449,-101.015,-43.262,178.813,5.930,149.412
C09979=1153.444,-100.765,-43.272,178.815,5.930,149.412
C09980=1153.438,-100.515,-43.281,178.817,5.930,149.411
C09981=1153.433,-100.265,-43.290,178.819,5.931,149.411
C09982=1153.428,-100.015,-43.299,178.821,5.931,149.410
C09983=1153.422,-99.766,-43.309,178.823,5.932,149.410
C09984=1153.417,-99.516,-43.318,178.826,5.932,149.409
C09985=1153.412,-99.266,-43.327,178.827,5.932,149.409
C09986=1153.406,-99.016,-43.337,178.830,5.933,149.408
C09987=1153.401,-98.768,-43.346,178.831,5.933,149.408
C09988=1153.395,-98.517,-43.355,178.834,5.933,149.407
C09989=1153.390,-98.267,-43.364,178.836,5.934,149.407
C09990=1153.385,-98.018,-43.374,178.838,5.934,149.406
C09991=1153.379,-97.768,-43.383,178.840,5.935,149.405
C09992=1153.374,-97.518,-43.393,178.842,5.934,149.405
C09993=1153.369,-97.268,-43.402,178.844,5.935,149.404
C09994=1153.363,-97.018,-43.412,178.847,5.936,149.404
C09995=1153.358,-96.768,-43.421,178.848,5.936,149.403
C09996=1153.353,-96.519,-43.431,178.850,5.936,149.403
//INST
///DATE 2021/06/25 14:31
///ATTR SC,RW,RJ
////FRAME ROBOT
///GROUP1 RB1
NOP
MOVL C00000 V=800.0 PL=0
MOVL C00001 V=800.0 PL=0
MOVL C00002 V=800.0 PL=0
MOVL C00003 V=800.0 PL=0
MOVL C00004 V=800.0 PL=0
MOVL C00005 V=800.0 PL=0
MOVL C00006 V=800.0 PL=0
MOVL C00007 V=800.0 PL=0
MOVL C00008 V=800.0 PL=0
MOVL C00009 V=800.0 PL=0
MOVL C00010 V=800.0 PL=0
MOVL C00011 V=800.0 PL=0
MOVL C00012 V=800.0 PL=0
MOVL C00013 V=800.0 PL=0
MOVL C00014 V=800.0 PL=0
MOVL C00015 V=800.0 PL=0
MOVL C00016 V=800.0 PL=0
MOVL C00017 V=800.0 PL=0
MOVL C00018 V=800.0 PL=0
MOVL C00019 V=800.0 PL=0
MOVL C00020 V=800.0 PL=0
MOVL C00021 V=800.0 PL=0
MOVL C00022 V=800.0 PL=0
MOVL C00023 V=800.0 PL=0
MOVL C00024 V=800.0 PL=0
MOVL C00025 V=800.0 PL=0
MOVL C00026 V=800.0 PL=0
MOVL C00027 V=800.0 PL=0
MOVL C00028 V=800.0 PL=0
MOVL C00029 V=800.0 PL=0
MOVL C00030 V=800.0 PL=0
MOVL C00031 V=800.0 PL=0
MOVL C00032 V=800.0 PL=0
MOVL C00033 V=800.0 PL=0
MOVL C00034 V=800.0 PL=0
MOVL C00035 V=800.0 PL=0
MOVL C00036 V=800.0 PL=0
MOVL C00037 V=800.0 PL=0
MOVL C00038 V=800.0 PL=0
MOVL C00039 V=800.0 PL=0
MOVL C00040 V=800.0 PL=0
MOVL C00041 V=800.0 PL=0
MOVL C00042 V=800.0 PL=0
MOVL C00043 V=800.0 PL=0
MOVL C00044 V=800.0 PL=0
MOVL C00045 V=800.0 PL=0
MOVL C00046 V=800.0 PL=0
MOVL C00047 V=800.0 PL=0
MOVL C00048 V=800.0 PL=0
MOVL C00049 V=800.0 PL=0
MOVL C00050 V=800.0 PL=0
MOVL C00051 V=800.0 PL=0
MOVL C00052 V=800.0 PL=0
MOVL C00053 V=800.0 PL=0
MOVL C00054 V=800.0 PL=0
MOVL C00055 V=800.0 PL=0
MOVL C00056 V=800.0 PL=0
MOVL C00057 V=800.0 PL=0
MOVL C00058 V=800.0 PL=0
MOVL C00059 V=800.0 PL=0
MOVL C00060 V=800.0 PL=0
MOVL C00061 V=800.0 PL=0
MOVL C00062 V=800.0 PL=0
MOVL C00063 V=800.0 PL=0
MOVL C00064 V=800.0 PL=0
MOVL C00065 V=800.0 PL=0
MOVL C00066 V=800.0 PL=0
MOVL C00067 V=800.0 PL=0
MOVL C00068 V=800.0 PL=0
MOVL C00069 V=800.0 PL=0
MOVL C00070 V=800.0 PL=0
MOVL C00071 V=800.0 PL=0
MOVL C00072 V=800.0 PL=0
MOVL C00073 V=800.0 PL=0
MOVL C00074 V=800.0 PL=0
MOVL C00075 V=800.0 PL=0
MOVL C00076 V=800.0 PL=0
MOVL C00077 V=800.0 PL=0
MOVL C00078 V=800.0 PL=0
MOVL C00079 V=800.0 PL=0
MOVL C00080 V=800.0 PL=0
MOVL C00081 V=800.0 PL=0
MOVL C00082 V=800.0 PL=0
MOVL C00083 V=800.0 PL=0
MOVL C00084 V=800.0 PL=0
MOVL C00085 V=800.0 PL=0
MOVL C00086 V=800.0 PL=0
MOVL C00087 V=800.0 PL=0
MOVL C00088 V=800.0 PL=0
MOVL C00089 V=800.0 PL=0
MOVL C00090 V=800.0 PL=0
MOVL C00091 V=800.0 PL=0
MOVL C00092 V=800.0 PL=0
MOVL C00093 V=800.0 PL=0
MOVL C00094 V=800.0 PL=0
MOVL C00095 V=800.0 PL=0
MOVL C00096 V=800.0 PL=0
MOVL C00097 V=800.0 PL=0
MOVL C00098 V=800.0 PL=0
MOVL C00099 V=800.0 PL=0
MOVL C00100 V=800.0 PL=0
MOVL C00101 V=800.0 PL=0
MOVL C00102 V=800.0 PL=0
MOVL C00103 V=800.0 PL=0
MOVL C00104 V=800.0 PL=0
MOVL C00105 V=800.0 PL=0
MOVL C00106 V=800.0 PL=0
MOVL C00107 V=800.0 PL=0
MOVL C00108 V=800.0 PL=0
MOVL C00109 V=800.0 PL=0
MOVL C00110 V=800.0 PL=0
MOVL C00111 V=800.0 PL=0
MOVL C00112 V=800.0 PL=0
MOVL C00113 V=800.0 PL=0
MOVL C00114 V=800.0 PL=0
MOVL C00115 V=800.0 PL=0
MOVL C00116 V=800.0 PL=0
MOVL C00117 V=800.0 PL=0
MOVL C00118 V=800.0 PL=0
MOVL C00119 V=800.0 PL=0
MOVL C00120 V=800.0 PL=0
MOVL C00121 V=800.0 PL=0
MOVL C00122 V=800.0 PL=0
MOVL C00123 V=800.0 PL=0
MOVL C00124 V=800.0 PL=0
MOVL C00125 V=800.0 PL=0
MOVL C00126 V=800.0 PL=0
MOVL C00127 V=800.0 PL=0
MOVL C00128 V=800.0 PL=0
MOVL C00129 V=800.0 PL=0
MOVL C00130 V=800.0 PL=0
MOVL C00131 V=800.0 PL=0
MOVL C00132 V=800.0 PL=0
MOVL C00133 V=800.0 PL=0
MOVL C00134 V=800.0 PL=0
MOVL C00135 V=800.0 PL=0
MOVL C00136 V=800.0 PL=0
MOVL C00137 V=800.0 PL=0
MOVL C00138 V=800.0 PL=0
MOVL C00139 V=800.0 PL=0
MOVL C00140 V=800.0 PL=0
MOVL C00141 V=800.0 PL=0
MOVL C00142 V=800.0 PL=0
MOVL C00143 V=800.0 PL=0
MOVL C00144 V=800.0 PL=0
MOVL C00145 V=800.0 PL=0
MOVL C00146 V=800.0 PL=0
MOVL C00147 V=800.0 PL=0
MOVL C00148 V=800.0 PL=0
MOVL C00149 V=800.0 PL=0
MOVL C00150 V=800.0 PL=0
MOVL C00151 V=800.0 PL=0
MOVL C00152 V=800.0 PL=0
MOVL C00153 V=800.0 PL=0
MOVL C00154 V=800.0 PL=0
MOVL C00155 V=800.0 PL=0
MOVL C00156 V=800.0 PL=0
MOVL C00157 V=800.0 PL=0
MOVL C00158 V=800.0 PL=0
MOVL C00159 V=800.0 PL=0
MOVL C00160 V=800.0 PL=0
MOVL C00161 V=800.0 PL=0
MOVL C00162 V=800.0 PL=0
MOVL C00163 V=800.0 PL=0
MOVL C00164 V=800.0 PL=0
MOVL C00165 V=800.0 PL=0
MOVL C00166 V=800.0 PL=0
MOVL C00167 V=800.0 PL=0
MOVL C00168 V=800.0 PL=0
MOVL C00169 V=800.0 PL=0
MOVL C00170 V=800.0 PL=0
MOVL C00171 V=800.0 PL=0
MOVL C00172 V=800.0 PL=0
MOVL C00173 V=800.0 PL=0
MOVL C00174 V=800.0 PL=0
MOVL C00175 V=800.0 PL=0
MOVL C00176 V=800.0 PL=0
MOVL C00177 V=800.0 PL=0
MOVL C00178 V=800.0 PL=0
MOVL C00179 V=800.0 PL=0
MOVL C00180 V=800.0 PL=0
MOVL C00181 V=800.0 PL=0
MOVL C00182 V=800.0 PL=0
MOVL C00183 V=800.0 PL=0
MOVL C00184 V=800.0 PL=0
MOVL C00185 V=800.0 PL=0
MOVL C00186 V=800.0 PL=0
MOVL C00187 V=800.0 PL=0
MOVL C00188 V=800.0 PL=0
MOVL C00189 V=800.0 PL=0
MOVL C00190 V=800.0 PL=0
MOVL C00191 V=800.0 PL=0
MOVL C00192 V=800.0 PL=0
MOVL C00193 V=800.0 PL=0
MOVL C00194 V=800.0 PL=0
MOVL C00195 V=800.0 PL=0
MOVL C00196 V=800.0 PL=0
MOVL C00197 V=800.0 PL=0
MOVL C00198 V=800.0 PL=0
MOVL C00199 V=800.0 PL=0
MOVL C00200 V=800.0 PL=0
MOVL C00201 V=800.0 PL=0
MOVL C00202 V=800.0 PL=0
MOVL C00203 V=800.0 PL=0
MOVL C00204 V=800.0 PL=0
MOVL C00205 V=800.0 PL=0
MOVL C00206 V=800.0 PL=0
MOVL C00207 V=800.0 PL=0
MOVL C00208 V=800.0 PL=0
MOVL C00209 V=800.0 PL=0
MOVL C00210 V=800.0 PL=0
MOVL C00211 V=800.0 PL=0
MOVL C00212 V=800.0 PL=0
MOVL C00213 V=800.0 PL=0
MOVL C00214 V=800.0 PL=0
MOVL C00215 V=800.0 PL=0
MOVL C00216 V=800.0 PL=0
MOVL C00217 V=800.0 PL=0
MOVL C00218 V=800.0 PL=0
MOVL C00219 V=800.0 PL=0
MOVL C00220 V=800.0 PL=0
MOVL C00221 V=800.0 PL=0
MOVL C00222 V=800.0 PL=0
MOVL C00223 V=800.0 PL=0
MOVL C00224 V=800.0 PL=0
MOVL C00225 V=800.0 PL=0
MOVL C00226 V=800.0 PL=0
MOVL C00227 V=800.0 PL=0
MOVL C00228 V=800.0 PL=0
MOVL C00229 V=800.0 PL=0
MOVL C00230 V=800.0 PL=0
MOVL C00231 V=800.0 PL=0
MOVL C00232 V=800.0 PL=0
MOVL C00233 V=800.0 PL=0
MOVL C00234 V=800.0 PL=0
MOVL C00235 V=800.0 PL=0
MOVL C00236 V=800.0 PL=0
MOVL C00237 V=800.0 PL=0
MOVL C00238 V=800.0 PL=0
MOVL C00239 V=800.0 PL=0
MOVL C00240 V=800.0 PL=0
MOVL C00241 V=800.0 PL=0
MOVL C00242 V=800.0 PL=0
MOVL C00243 V=800.0 PL=0
MOVL C00244 V=800.0 PL=0
MOVL C00245 V=800.0 PL=0
MOVL C00246 V=800.0 PL=0
MOVL C00247 V=800.0 PL=0
MOVL C00248 V=800.0 PL=0
MOVL C00249 V=800.0 PL=0
MOVL C00250 V=800.0 PL=0
MOVL C00251 V=800.0 PL=0
MOVL C00252 V=800.0 PL=0
MOVL C00253 V=800.0 PL=0
MOVL C00254 V=800.0 PL=0
MOVL C00255 V=800.0 PL=0
MOVL C00256 V=800.0 PL=0
MOVL C00257 V=800.0 PL=0
MOVL C00258 V=800.0 PL=0
MOVL C00259 V=800.0 PL=0
MOVL C00260 V=800.0 PL=0
MOVL C00261 V=800.0 PL=0
MOVL C00262 V=800.0 PL=0
MOVL C00263 V=800.0 PL=0
MOVL C00264 V=800.0 PL=0
MOVL C00265 V=800.0 PL=0
MOVL C00266 V=800.0 PL=0
MOVL C00267 V=800.0 PL=0
MOVL C00268 V=800.0 PL=0
MOVL C00269 V=800.0 PL=0
MOVL C00270 V=800.0 PL=0
MOVL C00271 V=800.0 PL=0
MOVL C00272 V=800.0 PL=0
MOVL C00273 V=800.0 PL=0
MOVL C00274 V=800.0 PL=0
MOVL C00275 V=800.0 PL=0
MOVL C00276 V=800.0 PL=0
MOVL C00277 V=800.0 PL=0
MOVL C00278 V=800.0 PL=0
MOVL C00279 V=800.0 PL=0
MOVL C00280 V=800.0 PL=0
MOVL C00281 V=800.0 PL=0
MOVL C00282 V=800.0 PL=0
MOVL C00283 V=800.0 PL=0
MOVL C00284 V=800.0 PL=0
MOVL C00285 V=800.0 PL=0
MOVL C00286 V=800.0 PL=0
MOVL C00287 V=800.0 PL=0
MOVL C00288 V=800.0 PL=0
MOVL C00289 V=800.0 PL=0
MOVL C00290 V=800.0 PL=0
MOVL C00291 V=800.0 PL=0
MOVL C00292 V=800.0 PL=0
MOVL C00293 V=800.0 PL=0
MOVL C00294 V=800.0 PL=0
MOVL C00295 V=800.0 PL=0
MOVL C00296 V=800.0 PL=0
MOVL C00297 V=800.0 PL=0
MOVL C00298 V=800.0 PL=0
MOVL C00299 V=800.0 PL=0
MOVL C00300 V=800.0 PL=0
MOVL C00301 V=800.0 PL=0
MOVL C00302 V=800.0 PL=0
MOVL C00303 V=800.0 PL=0
MOVL C00304 V=800.0 PL=0
MOVL C00305 V=800.0 PL=0
MOVL C00306 V=800.0 PL=0
MOVL C00307 V=800.0 PL=0
MOVL C00308 V=800.0 PL=0
MOVL C00309 V=800.0 PL=0
MOVL C00310 V=800.0 PL=0
MOVL C00311 V=800.0 PL=0
MOVL C00312 V=800.0 PL=0
MOVL C00313 V=800.0 PL=0
MOVL C00314 V=800.0 PL=0
MOVL C00315 V=800.0 PL=0
MOVL C00316 V=800.0 PL=0
MOVL C00317 V=800.0 PL=0
MOVL C00318 V=800.0 PL=0
MOVL C00319 V=800.0 PL=0
MOVL C00320 V=800.0 PL=0
MOVL C00321 V=800.0 PL=0
MOVL C00322 V=800.0 PL=0
MOVL C00323 V=800.0 PL=0
MOVL C00324 V=800.0 PL=0
MOVL C00325 V=800.0 PL=0
MOVL C00326 V=800.0 PL=0
MOVL C00327 V=800.0 PL=0
MOVL C00328 V=800.0 PL=0
MOVL C00329 V=800.0 PL=0
MOVL C00330 V=800.0 PL=0
MOVL C00331 V=800.0 PL=0
MOVL C00332 V=800.0 PL=0
MOVL C00333 V=800.0 PL=0
MOVL C00334 V=800.0 PL=0
MOVL C00335 V=800.0 PL=0
MOVL C00336 V=800.0 PL=0
MOVL C00337 V=800.0 PL=0
MOVL C00338 V=800.0 PL=0
MOVL C00339 V=800.0 PL=0
MOVL C00340 V=800.0 PL=0
MOVL C00341 V=800.0 PL=0
MOVL C00342 V=800.0 PL=0
MOVL C00343 V=800.0 PL=0
MOVL C00344 V=800.0 PL=0
MOVL C00345 V=800.0 PL=0
MOVL C00346 V=800.0 PL=0
MOVL C00347 V=800.0 PL=0
MOVL C00348 V=800.0 PL=0
MOVL C00349 V=800.0 PL=0
MOVL C00350 V=800.0 PL=0
MOVL C00351 V=800.0 PL=0
MOVL C00352 V=800.0 PL=0
MOVL C00353 V=800.0 PL=0
MOVL C00354 V=800.0 PL=0
MOVL C00355 V=800.0 PL=0
MOVL C00356 V=800.0 PL=0
MOVL C00357 V=800.0 PL=0
MOVL C00358 V=800.0 PL=0
MOVL C00359 V=800.0 PL=0
MOVL C00360 V=800.0 PL=0
MOVL C00361 V=800.0 PL=0
MOVL C00362 V=800.0 PL=0
MOVL C00363 V=800.0 PL=0
MOVL C00364 V=800.0 PL=0
MOVL C00365 V=800.0 PL=0
MOVL C00366 V=800.0 PL=0
MOVL C00367 V=800.0 PL=0
MOVL C00368 V=800.0 PL=0
MOVL C00369 V=800.0 PL=0
MOVL C00370 V=800.0 PL=0
MOVL C00371 V=800.0 PL=0
MOVL C00372 V=800.0 PL=0
MOVL C00373 V=800.0 PL=0
MOVL C00374 V=800.0 PL=0
MOVL C00375 V=800.0 PL=0
MOVL C00376 V=800.0 PL=0
MOVL C00377 V=800.0 PL=0
MOVL C00378 V=800.0 PL=0
MOVL C00379 V=800.0 PL=0
MOVL C00380 V=800.0 PL=0
MOVL C00381 V=800.0 PL=0
MOVL C00382 V=800.0 PL=0
MOVL C00383 V=800.0 PL=0
MOVL C00384 V=800.0 PL=0
MOVL C00385 V=800.0 PL=0
MOVL C00386 V=800.0 PL=0
MOVL C00387 V=800.0 PL=0
MOVL C00388 V=800.0 PL=0
MOVL C00389 V=800.0 PL=0
MOVL C00390 V=800.0 PL=0
MOVL C00391 V=800.0 PL=0
MOVL C00392 V=800.0 PL=0
MOVL C00393 V=800.0 PL=0
MOVL C00394 V=800.0 PL=0
MOVL C00395 V=800.0 PL=0
MOVL C00396 V=800.0 PL=0
MOVL C00397 V=800.0 PL=0
MOVL C00398 V=800.0 PL=0
MOVL C00399 V=800.0 PL=0
MOVL C00400 V=800.0 PL=0
MOVL C00401 V=800.0 PL=0
MOVL C00402 V=800.0 PL=0
MOVL C00403 V=800.0 PL=0
MOVL C00404 V=800.0 PL=0
MOVL C00405 V=800.0 PL=0
MOVL C00406 V=800.0 PL=0
MOVL C00407 V=800.0 PL=0
MOVL C00408 V=800.0 PL=0
MOVL C00409 V=800.0 PL=0
MOVL C00410 V=800.0 PL=0
MOVL C00411 V=800.0 PL=0
MOVL C00412 V=800.0 PL=0
MOVL C00413 V=800.0 PL=0
MOVL C00414 V=800.0 PL=0
MOVL C00415 V=800.0 PL=0
MOVL C00416 V=800.0 PL=0
MOVL C00417 V=800.0 PL=0
MOVL C00418 V=800.0 PL=0
MOVL C00419 V=800.0 PL=0
MOVL C00420 V=800.0 PL=0
MOVL C00421 V=800.0 PL=0
MOVL C00422 V=800.0 PL=0
MOVL C00423 V=800.0 PL=0
MOVL C00424 V=800.0 PL=0
MOVL C00425 V=800.0 PL=0
MOVL C00426 V=800.0 PL=0
MOVL C00427 V=800.0 PL=0
MOVL C00428 V=800.0 PL=0
MOVL C00429 V=800.0 PL=0
MOVL C00430 V=800.0 PL=0
MOVL C00431 V=800.0 PL=0
MOVL C00432 V=800.0 PL=0
MOVL C00433 V=800.0 PL=0
MOVL C00434 V=800.0 PL=0
MOVL C00435 V=800.0 PL=0
MOVL C00436 V=800.0 PL=0
MOVL C00437 V=800.0 PL=0
MOVL C00438 V=800.0 PL=0
MOVL C00439 V=800.0 PL=0
MOVL C00440 V=800.0 PL=0
MOVL C00441 V=800.0 PL=0
MOVL C00442 V=800.0 PL=0
MOVL C00443 V=800.0 PL=0
MOVL C00444 V=800.0 PL=0
MOVL C00445 V=800.0 PL=0
MOVL C00446 V=800.0 PL=0
MOVL C00447 V=800.0 PL=0
MOVL C00448 V=800.0 PL=0
MOVL C00449 V=800.0 PL=0
MOVL C00450 V=800.0 PL=0
MOVL C00451 V=800.0 PL=0
MOVL C00452 V=800.0 PL=0
MOVL C00453 V=800.0 PL=0
MOVL C00454 V=800.0 PL=0
MOVL C00455 V=800.0 PL=0
MOVL C00456 V=800.0 PL=0
MOVL C00457 V=800.0 PL=0
MOVL C00458 V=800.0 PL=0
MOVL C00459 V=800.0 PL=0
MOVL C00460 V=800.0 PL=0
MOVL C00461 V=800.0 PL=0
MOVL C00462 V=800.0 PL=0
MOVL C00463 V=800.0 PL=0
MOVL C00464 V=800.0 PL=0
MOVL C00465 V=800.0 PL=0
MOVL C00466 V=800.0 PL=0
MOVL C00467 V=800.0 PL=0
MOVL C00468 V=800.0 PL=0
MOVL C00469 V=800.0 PL=0
MOVL C00470 V=800.0 PL=0
MOVL C00471 V=800.0 PL=0
MOVL C00472 V=800.0 PL=0
MOVL C00473 V=800.0 PL=0
MOVL C00474 V=800.0 PL=0
MOVL C00475 V=800.0 PL=0
MOVL C00476 V=800.0 PL=0
MOVL C00477 V=800.0 PL=0
MOVL C00478 V=800.0 PL=0
MOVL C00479 V=800.0 PL=0
MOVL C00480 V=800.0 PL=0
MOVL C00481 V=800.0 PL=0
MOVL C00482 V=800.0 PL=0
MOVL C00483 V=800.0 PL=0
MOVL C00484 V=800.0 PL=0
MOVL C00485 V=800.0 PL=0
MOVL C00486 V=800.0 PL=0
MOVL C00487 V=800.0 PL=0
MOVL C00488 V=800.0 PL=0
MOVL C00489 V=800.0 PL=0
MOVL C00490 V=800.0 PL=0
MOVL C00491 V=800.0 PL=0
MOVL C00492 V=800.0 PL=0
MOVL C00493 V=800.0 PL=0
MOVL C00494 V=800.0 PL=0
MOVL C00495 V=800.0 PL=0
MOVL C00496 V=800.0 PL=0
MOVL C00497 V=800.0 PL=0
MOVL C00498 V=800.0 PL=0
MOVL C00499 V=800.0 PL=0
MOVL C00500 V=800.0 PL=0
MOVL C00501 V=800.0 PL=0
MOVL C00502 V=800.0 PL=0
MOVL C00503 V=800.0 PL=0
MOVL C00504 V=800.0 PL=0
MOVL C00505 V=800.0 PL=0
MOVL C00506 V=800.0 PL=0
MOVL C00507 V=800.0 PL=0
MOVL C00508 V=800.0 PL=0
MOVL C00509 V=800.0 PL=0
MOVL C00510 V=800.0 PL=0
MOVL C00511 V=800.0 PL=0
MOVL C00512 V=800.0 PL=0
MOVL C00513 V=800.0 PL=0
MOVL C00514 V=800.0 PL=0
MOVL C00515 V=800.0 PL=0
MOVL C00516 V=800.0 PL=0
MOVL C00517 V=800.0 PL=0
MOVL C00518 V=800.0 PL=0
MOVL C00519 V=800.0 PL=0
MOVL C00520 V=800.0 PL=0
MOVL C00521 V=800.0 PL=0
MOVL C00522 V=800.0 PL=0
MOVL C00523 V=800.0 PL=0
MOVL C00524 V=800.0 PL=0
MOVL C00525 V=800.0 PL=0
MOVL C00526 V=800.0 PL=0
MOVL C00527 V=800.0 PL=0
MOVL C00528 V=800.0 PL=0
MOVL C00529 V=800.0 PL=0
MOVL C00530 V=800.0 PL=0
MOVL C00531 V=800.0 PL=0
MOVL C00532 V=800.0 PL=0
MOVL C00533 V=800.0 PL=0
MOVL C00534 V=800.0 PL=0
MOVL C00535 V=800.0 PL=0
MOVL C00536 V=800.0 PL=0
MOVL C00537 V=800.0 PL=0
MOVL C00538 V=800.0 PL=0
MOVL C00539 V=800.0 PL=0
MOVL C00540 V=800.0 PL=0
MOVL C00541 V=800.0 PL=0
MOVL C00542 V=800.0 PL=0
MOVL C00543 V=800.0 PL=0
MOVL C00544 V=800.0 PL=0
MOVL C00545 V=800.0 PL=0
MOVL C00546 V=800.0 PL=0
MOVL C00547 V=800.0 PL=0
MOVL C00548 V=800.0 PL=0
MOVL C00549 V=800.0 PL=0
MOVL C00550 V=800.0 PL=0
MOVL C00551 V=800.0 PL=0
MOVL C00552 V=800.0 PL=0
MOVL C00553 V=800.0 PL=0
MOVL C00554 V=800.0 PL=0
MOVL C00555 V=800.0 PL=0
MOVL C00556 V=800.0 PL=0
MOVL C00557 V=800.0 PL=0
MOVL C00558 V=800.0 PL=0
MOVL C00559 V=800.0 PL=0
MOVL C00560 V=800.0 PL=0
MOVL C00561 V=800.0 PL=0
MOVL C00562 V=800.0 PL=0
MOVL C00563 V=800.0 PL=0
MOVL C00564 V=800.0 PL=0
MOVL C00565 V=800.0 PL=0
MOVL C00566 V=800.0 PL=0
MOVL C00567 V=800.0 PL=0
MOVL C00568 V=800.0 PL=0
MOVL C00569 V=800.0 PL=0
MOVL C00570 V=800.0 PL=0
MOVL C00571 V=800.0 PL=0
MOVL C00572 V=800.0 PL=0
MOVL C00573 V=800.0 PL=0
MOVL C00574 V=800.0 PL=0
MOVL C00575 V=800.0 PL=0
MOVL C00576 V=800.0 PL=0
MOVL C00577 V=800.0 PL=0
MOVL C00578 V=800.0 PL=0
MOVL C00579 V=800.0 PL=0
MOVL C00580 V=800.0 PL=0
MOVL C00581 V=800.0 PL=0
MOVL C00582 V=800.0 PL=0
MOVL C00583 V=800.0 PL=0
MOVL C00584 V=800.0 PL=0
MOVL C00585 V=800.0 PL=0
MOVL C00586 V=800.0 PL=0
MOVL C00587 V=800.0 PL=0
MOVL C00588 V=800.0 PL=0
MOVL C00589 V=800.0 PL=0
MOVL C00590 V=800.0 PL=0
MOVL C00591 V=800.0 PL=0
MOVL C00592 V=800.0 PL=0
MOVL C00593 V=800.0 PL=0
MOVL C00594 V=800.0 PL=0
MOVL C00595 V=800.0 PL=0
MOVL C00596 V=800.0 PL=0
MOVL C00597 V=800.0 PL=0
MOVL C00598 V=800.0 PL=0
MOVL C00599 V=800.0 PL=0
MOVL C00600 V=800.0 PL=0
MOVL C00601 V=800.0 PL=0
MOVL C00602 V=800.0 PL=0
MOVL C00603 V=800.0 PL=0
MOVL C00604 V=800.0 PL=0
MOVL C00605 V=800.0 PL=0
MOVL C00606 V=800.0 PL=0
MOVL C00607 V=800.0 PL=0
MOVL C00608 V=800.0 PL=0
MOVL C00609 V=800.0 PL=0
MOVL C00610 V=800.0 PL=0
MOVL C00611 V=800.0 PL=0
MOVL C00612 V=800.0 PL=0
MOVL C00613 V=800.0 PL=0
MOVL C00614 V=800.0 PL=0
MOVL C00615 V=800.0 PL=0
MOVL C00616 V=800.0 PL=0
MOVL C00617 V=800.0 PL=0
MOVL C00618 V=800.0 PL=0
MOVL C00619 V=800.0 PL=0
MOVL C00620 V=800.0 PL=0
MOVL C00621 V=800.0 PL=0
MOVL C00622 V=800.0 PL=0
MOVL C00623 V=800.0 PL=0
MOVL C00624 V=800.0 PL=0
MOVL C00625 V=800.0 PL=0
MOVL C00626 V=800.0 PL=0
MOVL C00627 V=800.0 PL=0
MOVL C00628 V=800.0 PL=0
MOVL C00629 V=800.0 PL=0
MOVL C00630 V=800.0 PL=0
MOVL C00631 V=800.0 PL=0
MOVL C00632 V=800.0 PL=0
MOVL C00633 V=800.0 PL=0
MOVL C00634 V=800.0 PL=0
MOVL C00635 V=800.0 PL=0
MOVL C00636 V=800.0 PL=0
MOVL C00637 V=800.0 PL=0
MOVL C00638 V=800.0 PL=0
MOVL C00639 V=800.0 PL=0
MOVL C00640 V=800.0 PL=0
MOVL C00641 V=800.0 PL=0
MOVL C00642 V=800.0 PL=0
MOVL C00643 V=800.0 PL=0
MOVL C00644 V=800.0 PL=0
MOVL C00645 V=800.0 PL=0
MOVL C00646 V=800.0 PL=0
MOVL C00647 V=800.0 PL=0
MOVL C00648 V=800.0 PL=0
MOVL C00649 V=800.0 PL=0
MOVL C00650 V=800.0 PL=0
MOVL C00651 V=800.0 PL=0
MOVL C00652 V=800.0 PL=0
MOVL C00653 V=800.0 PL=0
MOVL C00654 V=800.0 PL=0
MOVL C00655 V=800.0 PL=0
MOVL C00656 V=800.0 PL=0
MOVL C00657 V=800.0 PL=0
MOVL C00658 V=800.0 PL=0
MOVL C00659 V=800.0 PL=0
MOVL C00660 V=800.0 PL=0
MOVL C00661 V=800.0 PL=0
MOVL C00662 V=800.0 PL=0
MOVL C00663 V=800.0 PL=0
MOVL C00664 V=800.0 PL=0
MOVL C00665 V=800.0 PL=0
MOVL C00666 V=800.0 PL=0
MOVL C00667 V=800.0 PL=0
MOVL C00668 V=800.0 PL=0
MOVL C00669 V=800.0 PL=0
MOVL C00670 V=800.0 PL=0
MOVL C00671 V=800.0 PL=0
MOVL C00672 V=800.0 PL=0
MOVL C00673 V=800.0 PL=0
MOVL C00674 V=800.0 PL=0
MOVL C00675 V=800.0 PL=0
MOVL C00676 V=800.0 PL=0
MOVL C00677 V=800.0 PL=0
MOVL C00678 V=800.0 PL=0
MOVL C00679 V=800.0 PL=0
MOVL C00680 V=800.0 PL=0
MOVL C00681 V=800.0 PL=0
MOVL C00682 V=800.0 PL=0
MOVL C00683 V=800.0 PL=0
MOVL C00684 V=800.0 PL=0
MOVL C00685 V=800.0 PL=0
MOVL C00686 V=800.0 PL=0
MOVL C00687 V=800.0 PL=0
MOVL C00688 V=800.0 PL=0
MOVL C00689 V=800.0 PL=0
MOVL C00690 V=800.0 PL=0
MOVL C00691 V=800.0 PL=0
MOVL C00692 V=800.0 PL=0
MOVL C00693 V=800.0 PL=0
MOVL C00694 V=800.0 PL=0
MOVL C00695 V=800.0 PL=0
MOVL C00696 V=800.0 PL=0
MOVL C00697 V=800.0 PL=0
MOVL C00698 V=800.0 PL=0
MOVL C00699 V=800.0 PL=0
MOVL C00700 V=800.0 PL=0
MOVL C00701 V=800.0 PL=0
MOVL C00702 V=800.0 PL=0
MOVL C00703 V=800.0 PL=0
MOVL C00704 V=800.0 PL=0
MOVL C00705 V=800.0 PL=0
MOVL C00706 V=800.0 PL=0
MOVL C00707 V=800.0 PL=0
MOVL C00708 V=800.0 PL=0
MOVL C00709 V=800.0 PL=0
MOVL C00710 V=800.0 PL=0
MOVL C00711 V=800.0 PL=0
MOVL C00712 V=800.0 PL=0
MOVL C00713 V=800.0 PL=0
MOVL C00714 V=800.0 PL=0
MOVL C00715 V=800.0 PL=0
MOVL C00716 V=800.0 PL=0
MOVL C00717 V=800.0 PL=0
MOVL C00718 V=800.0 PL=0
MOVL C00719 V=800.0 PL=0
MOVL C00720 V=800.0 PL=0
MOVL C00721 V=800.0 PL=0
MOVL C00722 V=800.0 PL=0
MOVL C00723 V=800.0 PL=0
MOVL C00724 V=800.0 PL=0
MOVL C00725 V=800.0 PL=0
MOVL C00726 V=800.0 PL=0
MOVL C00727 V=800.0 PL=0
MOVL C00728 V=800.0 PL=0
MOVL C00729 V=800.0 PL=0
MOVL C00730 V=800.0 PL=0
MOVL C00731 V=800.0 PL=0
MOVL C00732 V=800.0 PL=0
MOVL C00733 V=800.0 PL=0
MOVL C00734 V=800.0 PL=0
MOVL C00735 V=800.0 PL=0
MOVL C00736 V=800.0 PL=0
MOVL C00737 V=800.0 PL=0
MOVL C00738 V=800.0 PL=0
MOVL C00739 V=800.0 PL=0
MOVL C00740 V=800.0 PL=0
MOVL C00741 V=800.0 PL=0
MOVL C00742 V=800.0 PL=0
MOVL C00743 V=800.0 PL=0
MOVL C00744 V=800.0 PL=0
MOVL C00745 V=800.0 PL=0
MOVL C00746 V=800.0 PL=0
MOVL C00747 V=800.0 PL=0
MOVL C00748 V=800.0 PL=0
MOVL C00749 V=800.0 PL=0
MOVL C00750 V=800.0 PL=0
MOVL C00751 V=800.0 PL=0
MOVL C00752 V=800.0 PL=0
MOVL C00753 V=800.0 PL=0
MOVL C00754 V=800.0 PL=0
MOVL C00755 V=800.0 PL=0
MOVL C00756 V=800.0 PL=0
MOVL C00757 V=800.0 PL=0
MOVL C00758 V=800.0 PL=0
MOVL C00759 V=800.0 PL=0
MOVL C00760 V=800.0 PL=0
MOVL C00761 V=800.0 PL=0
MOVL C00762 V=800.0 PL=0
MOVL C00763 V=800.0 PL=0
MOVL C00764 V=800.0 PL=0
MOVL C00765 V=800.0 PL=0
MOVL C00766 V=800.0 PL=0
MOVL C00767 V=800.0 PL=0
MOVL C00768 V=800.0 PL=0
MOVL C00769 V=800.0 PL=0
MOVL C00770 V=800.0 PL=0
MOVL C00771 V=800.0 PL=0
MOVL C00772 V=800.0 PL=0
MOVL C00773 V=800.0 PL=0
MOVL C00774 V=800.0 PL=0
MOVL C00775 V=800.0 PL=0
MOVL C00776 V=800.0 PL=0
MOVL C00777 V=800.0 PL=0
MOVL C00778 V=800.0 PL=0
MOVL C00779 V=800.0 PL=0
MOVL C00780 V=800.0 PL=0
MOVL C00781 V=800.0 PL=0
MOVL C00782 V=800.0 PL=0
MOVL C00783 V=800.0 PL=0
MOVL C00784 V=800.0 PL=0
MOVL C00785 V=800.0 PL=0
MOVL C00786 V=800.0 PL=0
MOVL C00787 V=800.0 PL=0
MOVL C00788 V=800.0 PL=0
MOVL C00789 V=800.0 PL=0
MOVL C00790 V=800.0 PL=0
MOVL C00791 V=800.0 PL=0
MOVL C00792 V=800.0 PL=0
MOVL C00793 V=800.0 PL=0
MOVL C00794 V=800.0 PL=0
MOVL C00795 V=800.0 PL=0
MOVL C00796 V=800.0 PL=0
MOVL C00797 V=800.0 PL=0
MOVL C00798 V=800.0 PL=0
MOVL C00799 V=800.0 PL=0
MOVL C00800 V=800.0 PL=0
MOVL C00801 V=800.0 PL=0
MOVL C00802 V=800.0 PL=0
MOVL C00803 V=800.0 PL=0
MOVL C00804 V=800.0 PL=0
MOVL C00805 V=800.0 PL=0
MOVL C00806 V=800.0 PL=0
MOVL C00807 V=800.0 PL=0
MOVL C00808 V=800.0 PL=0
MOVL C00809 V=800.0 PL=0
MOVL C00810 V=800.0 PL=0
MOVL C00811 V=800.0 PL=0
MOVL C00812 V=800.0 PL=0
MOVL C00813 V=800.0 PL=0
MOVL C00814 V=800.0 PL=0
MOVL C00815 V=800.0 PL=0
MOVL C00816 V=800.0 PL=0
MOVL C00817 V=800.0 PL=0
MOVL C00818 V=800.0 PL=0
MOVL C00819 V=800.0 PL=0
MOVL C00820 V=800.0 PL=0
MOVL C00821 V=800.0 PL=0
MOVL C00822 V=800.0 PL=0
MOVL C00823 V=800.0 PL=0
MOVL C00824 V=800.0 PL=0
MOVL C00825 V=800.0 PL=0
MOVL C00826 V=800.0 PL=0
MOVL C00827 V=800.0 PL=0
MOVL C00828 V=800.0 PL=0
MOVL C00829 V=800.0 PL=0
MOVL C00830 V=800.0 PL=0
MOVL C00831 V=800.0 PL=0
MOVL C00832 V=800.0 PL=0
MOVL C00833 V=800.0 PL=0
MOVL C00834 V=800.0 PL=0
MOVL C00835 V=800.0 PL=0
MOVL C00836 V=800.0 PL=0
MOVL C00837 V=800.0 PL=0
MOVL C00838 V=800.0 PL=0
MOVL C00839 V=800.0 PL=0
MOVL C00840 V=800.0 PL=0
MOVL C00841 V=800.0 PL=0
MOVL C00842 V=800.0 PL=0
MOVL C00843 V=800.0 PL=0
MOVL C00844 V=800.0 PL=0
MOVL C00845 V=800.0 PL=0
MOVL C00846 V=800.0 PL=0
MOVL C00847 V=800.0 PL=0
MOVL C00848 V=800.0 PL=0
MOVL C00849 V=800.0 PL=0
MOVL C00850 V=800.0 PL=0
MOVL C00851 V=800.0 PL=0
MOVL C00852 V=800.0 PL=0
MOVL C00853 V=800.0 PL=0
MOVL C00854 V=800.0 PL=0
MOVL C00855 V=800.0 PL=0
MOVL C00856 V=800.0 PL=0
MOVL C00857 V=800.0 PL=0
MOVL C00858 V=800.0 PL=0
MOVL C00859 V=800.0 PL=0
MOVL C00860 V=800.0 PL=0
MOVL C00861 V=800.0 PL=0
MOVL C00862 V=800.0 PL=0
MOVL C00863 V=800.0 PL=0
MOVL C00864 V=800.0 PL=0
MOVL C00865 V=800.0 PL=0
MOVL C00866 V=800.0 PL=0
MOVL C00867 V=800.0 PL=0
MOVL C00868 V=800.0 PL=0
MOVL C00869 V=800.0 PL=0
MOVL C00870 V=800.0 PL=0
MOVL C00871 V=800.0 PL=0
MOVL C00872 V=800.0 PL=0
MOVL C00873 V=800.0 PL=0
MOVL C00874 V=800.0 PL=0
MOVL C00875 V=800.0 PL=0
MOVL C00876 V=800.0 PL=0
MOVL C00877 V=800.0 PL=0
MOVL C00878 V=800.0 PL=0
MOVL C00879 V=800.0 PL=0
MOVL C00880 V=800.0 PL=0
MOVL C00881 V=800.0 PL=0
MOVL C00882 V=800.0 PL=0
MOVL C00883 V=800.0 PL=0
MOVL C00884 V=800.0 PL=0
MOVL C00885 V=800.0 PL=0
MOVL C00886 V=800.0 PL=0
MOVL C00887 V=800.0 PL=0
MOVL C00888 V=800.0 PL=0
MOVL C00889 V=800.0 PL=0
MOVL C00890 V=800.0 PL=0
MOVL C00891 V=800.0 PL=0
MOVL C00892 V=800.0 PL=0
MOVL C00893 V=800.0 PL=0
MOVL C00894 V=800.0 PL=0
MOVL C00895 V=800.0 PL=0
MOVL C00896 V=800.0 PL=0
MOVL C00897 V=800.0 PL=0
MOVL C00898 V=800.0 PL=0
MOVL C00899 V=800.0 PL=0
MOVL C00900 V=800.0 PL=0
MOVL C00901 V=800.0 PL=0
MOVL C00902 V=800.0 PL=0
MOVL C00903 V=800.0 PL=0
MOVL C00904 V=800.0 PL=0
MOVL C00905 V=800.0 PL=0
MOVL C00906 V=800.0 PL=0
MOVL C00907 V=800.0 PL=0
MOVL C00908 V=800.0 PL=0
MOVL C00909 V=800.0 PL=0
MOVL C00910 V=800.0 PL=0
MOVL C00911 V=800.0 PL=0
MOVL C00912 V=800.0 PL=0
MOVL C00913 V=800.0 PL=0
MOVL C00914 V=800.0 PL=0
MOVL C00915 V=800.0 PL=0
MOVL C00916 V=800.0 PL=0
MOVL C00917 V=800.0 PL=0
MOVL C00918 V=800.0 PL=0
MOVL C00919 V=800.0 PL=0
MOVL C00920 V=800.0 PL=0
MOVL C00921 V=800.0 PL=0
MOVL C00922 V=800.0 PL=0
MOVL C00923 V=800.0 PL=0
MOVL C00924 V=800.0 PL=0
MOVL C00925 V=800.0 PL=0
MOVL C00926 V=800.0 PL=0
MOVL C00927 V=800.0 PL=0
MOVL C00928 V=800.0 PL=0
MOVL C00929 V=800.0 PL=0
MOVL C00930 V=800.0 PL=0
MOVL C00931 V=800.0 PL=0
MOVL C00932 V=800.0 PL=0
MOVL C00933 V=800.0 PL=0
MOVL C00934 V=800.0 PL=0
MOVL C00935 V=800.0 PL=0
MOVL C00936 V=800.0 PL=0
MOVL C00937 V=800.0 PL=0
MOVL C00938 V=800.0 PL=0
MOVL C00939 V=800.0 PL=0
MOVL C00940 V=800.0 PL=0
MOVL C00941 V=800.0 PL=0
MOVL C00942 V=800.0 PL=0
MOVL C00943 V=800.0 PL=0
MOVL C00944 V=800.0 PL=0
MOVL C00945 V=800.0 PL=0
MOVL C00946 V=800.0 PL=0
MOVL C00947 V=800.0 PL=0
MOVL C00948 V=800.0 PL=0
MOVL C00949 V=800.0 PL=0
MOVL C00950 V=800.0 PL=0
MOVL C00951 V=800.0 PL=0
MOVL C00952 V=800.0 PL=0
MOVL C00953 V=800.0 PL=0
MOVL C00954 V=800.0 PL=0
MOVL C00955 V=800.0 PL=0
MOVL C00956 V=800.0 PL=0
MOVL C00957 V=800.0 PL=0
MOVL C00958 V=800.0 PL=0
MOVL C00959 V=800.0 PL=0
MOVL C00960 V=800.0 PL=0
MOVL C00961 V=800.0 PL=0
MOVL C00962 V=800.0 PL=0
MOVL C00963 V=800.0 PL=0
MOVL C00964 V=800.0 PL=0
MOVL C00965 V=800.0 PL=0
MOVL C00966 V=800.0 PL=0
MOVL C00967 V=800.0 PL=0
MOVL C00968 V=800.0 PL=0
MOVL C00969 V=800.0 PL=0
MOVL C00970 V=800.0 PL=0
MOVL C00971 V=800.0 PL=0
MOVL C00972 V=800.0 PL=0
MOVL C00973 V=800.0 PL=0
MOVL C00974 V=800.0 PL=0
MOVL C00975 V=800.0 PL=0
MOVL C00976 V=800.0 PL=0
MOVL C00977 V=800.0 PL=0
MOVL C00978 V=800.0 PL=0
MOVL C00979 V=800.0 PL=0
MOVL C00980 V=800.0 PL=0
MOVL C00981 V=800.0 PL=0
MOVL C00982 V=800.0 PL=0
MOVL C00983 V=800.0 PL=0
MOVL C00984 V=800.0 PL=0
MOVL C00985 V=800.0 PL=0
MOVL C00986 V=800.0 PL=0
MOVL C00987 V=800.0 PL=0
MOVL C00988 V=800.0 PL=0
MOVL C00989 V=800.0 PL=0
MOVL C00990 V=800.0 PL=0
MOVL C00991 V=800.0 PL=0
MOVL C00992 V=800.0 PL=0
MOVL C00993 V=800.0 PL=0
MOVL C00994 V=800.0 PL=0
MOVL C00995 V=800.0 PL=0
MOVL C00996 V=800.0 PL=0
MOVL C00997 V=800.0 PL=0
MOVL C00998 V=800.0 PL=0
MOVL C00999 V=800.0 PL=0
MOVL C01000 V=800.0 PL=0
MOVL C01001 V=800.0 PL=0
MOVL C01002 V=800.0 PL=0
MOVL C01003 V=800.0 PL=0
MOVL C01004 V=800.0 PL=0
MOVL C01005 V=800.0 PL=0
MOVL C01006 V=800.0 PL=0
MOVL C01007 V=800.0 PL=0
MOVL C01008 V=800.0 PL=0
MOVL C01009 V=800.0 PL=0
MOVL C01010 V=800.0 PL=0
MOVL C01011 V=800.0 PL=0
MOVL C01012 V=800.0 PL=0
MOVL C01013 V=800.0 PL=0
MOVL C01014 V=800.0 PL=0
MOVL C01015 V=800.0 PL=0
MOVL C01016 V=800.0 PL=0
MOVL C01017 V=800.0 PL=0
MOVL C01018 V=800.0 PL=0
MOVL C01019 V=800.0 PL=0
MOVL C01020 V=800.0 PL=0
MOVL C01021 V=800.0 PL=0
MOVL C01022 V=800.0 PL=0
MOVL C01023 V=800.0 PL=0
MOVL C01024 V=800.0 PL=0
MOVL C01025 V=800.0 PL=0
MOVL C01026 V=800.0 PL=0
MOVL C01027 V=800.0 PL=0
MOVL C01028 V=800.0 PL=0
MOVL C01029 V=800.0 PL=0
MOVL C01030 V=800.0 PL=0
MOVL C01031 V=800.0 PL=0
MOVL C01032 V=800.0 PL=0
MOVL C01033 V=800.0 PL=0
MOVL C01034 V=800.0 PL=0
MOVL C01035 V=800.0 PL=0
MOVL C01036 V=800.0 PL=0
MOVL C01037 V=800.0 PL=0
MOVL C01038 V=800.0 PL=0
MOVL C01039 V=800.0 PL=0
MOVL C01040 V=800.0 PL=0
MOVL C01041 V=800.0 PL=0
MOVL C01042 V=800.0 PL=0
MOVL C01043 V=800.0 PL=0
MOVL C01044 V=800.0 PL=0
MOVL C01045 V=800.0 PL=0
MOVL C01046 V=800.0 PL=0
MOVL C01047 V=800.0 PL=0
MOVL C01048 V=800.0 PL=0
MOVL C01049 V=800.0 PL=0
MOVL C01050 V=800.0 PL=0
MOVL C01051 V=800.0 PL=0
MOVL C01052 V=800.0 PL=0
MOVL C01053 V=800.0 PL=0
MOVL C01054 V=800.0 PL=0
MOVL C01055 V=800.0 PL=0
MOVL C01056 V=800.0 PL=0
MOVL C01057 V=800.0 PL=0
MOVL C01058 V=800.0 PL=0
MOVL C01059 V=800.0 PL=0
MOVL C01060 V=800.0 PL=0
MOVL C01061 V=800.0 PL=0
MOVL C01062 V=800.0 PL=0
MOVL C01063 V=800.0 PL=0
MOVL C01064 V=800.0 PL=0
MOVL C01065 V=800.0 PL=0
MOVL C01066 V=800.0 PL=0
MOVL C01067 V=800.0 PL=0
MOVL C01068 V=800.0 PL=0
MOVL C01069 V=800.0 PL=0
MOVL C01070 V=800.0 PL=0
MOVL C01071 V=800.0 PL=0
MOVL C01072 V=800.0 PL=0
MOVL C01073 V=800.0 PL=0
MOVL C01074 V=800.0 PL=0
MOVL C01075 V=800.0 PL=0
MOVL C01076 V=800.0 PL=0
MOVL C01077 V=800.0 PL=0
MOVL C01078 V=800.0 PL=0
MOVL C01079 V=800.0 PL=0
MOVL C01080 V=800.0 PL=0
MOVL C01081 V=800.0 PL=0
MOVL C01082 V=800.0 PL=0
MOVL C01083 V=800.0 PL=0
MOVL C01084 V=800.0 PL=0
MOVL C01085 V=800.0 PL=0
MOVL C01086 V=800.0 PL=0
MOVL C01087 V=800.0 PL=0
MOVL C01088 V=800.0 PL=0
MOVL C01089 V=800.0 PL=0
MOVL C01090 V=800.0 PL=0
MOVL C01091 V=800.0 PL=0
MOVL C01092 V=800.0 PL=0
MOVL C01093 V=800.0 PL=0
MOVL C01094 V=800.0 PL=0
MOVL C01095 V=800.0 PL=0
MOVL C01096 V=800.0 PL=0
MOVL C01097 V=800.0 PL=0
MOVL C01098 V=800.0 PL=0
MOVL C01099 V=800.0 PL=0
MOVL C01100 V=800.0 PL=0
MOVL C01101 V=800.0 PL=0
MOVL C01102 V=800.0 PL=0
MOVL C01103 V=800.0 PL=0
MOVL C01104 V=800.0 PL=0
MOVL C01105 V=800.0 PL=0
MOVL C01106 V=800.0 PL=0
MOVL C01107 V=800.0 PL=0
MOVL C01108 V=800.0 PL=0
MOVL C01109 V=800.0 PL=0
MOVL C01110 V=800.0 PL=0
MOVL C01111 V=800.0 PL=0
MOVL C01112 V=800.0 PL=0
MOVL C01113 V=800.0 PL=0
MOVL C01114 V=800.0 PL=0
MOVL C01115 V=800.0 PL=0
MOVL C01116 V=800.0 PL=0
MOVL C01117 V=800.0 PL=0
MOVL C01118 V=800.0 PL=0
MOVL C01119 V=800.0 PL=0
MOVL C01120 V=800.0 PL=0
MOVL C01121 V=800.0 PL=0
MOVL C01122 V=800.0 PL=0
MOVL C01123 V=800.0 PL=0
MOVL C01124 V=800.0 PL=0
MOVL C01125 V=800.0 PL=0
MOVL C01126 V=800.0 PL=0
MOVL C01127 V=800.0 PL=0
MOVL C01128 V=800.0 PL=0
MOVL C01129 V=800.0 PL=0
MOVL C01130 V=800.0 PL=0
MOVL C01131 V=800.0 PL=0
MOVL C01132 V=800.0 PL=0
MOVL C01133 V=800.0 PL=0
MOVL C01134 V=800.0 PL=0
MOVL C01135 V=800.0 PL=0
MOVL C01136 V=800.0 PL=0
MOVL C01137 V=800.0 PL=0
MOVL C01138 V=800.0 PL=0
MOVL C01139 V=800.0 PL=0
MOVL C01140 V=800.0 PL=0
MOVL C01141 V=800.0 PL=0
MOVL C01142 V=800.0 PL=0
MOVL C01143 V=800.0 PL=0
MOVL C01144 V=800.0 PL=0
MOVL C01145 V=800.0 PL=0
MOVL C01146 V=800.0 PL=0
MOVL C01147 V=800.0 PL=0
MOVL C01148 V=800.0 PL=0
MOVL C01149 V=800.0 PL=0
MOVL C01150 V=800.0 PL=0
MOVL C01151 V=800.0 PL=0
MOVL C01152 V=800.0 PL=0
MOVL C01153 V=800.0 PL=0
MOVL C01154 V=800.0 PL=0
MOVL C01155 V=800.0 PL=0
MOVL C01156 V=800.0 PL=0
MOVL C01157 V=800.0 PL=0
MOVL C01158 V=800.0 PL=0
MOVL C01159 V=800.0 PL=0
MOVL C01160 V=800.0 PL=0
MOVL C01161 V=800.0 PL=0
MOVL C01162 V=800.0 PL=0
MOVL C01163 V=800.0 PL=0
MOVL C01164 V=800.0 PL=0
MOVL C01165 V=800.0 PL=0
MOVL C01166 V=800.0 PL=0
MOVL C01167 V=800.0 PL=0
MOVL C01168 V=800.0 PL=0
MOVL C01169 V=800.0 PL=0
MOVL C01170 V=800.0 PL=0
MOVL C01171 V=800.0 PL=0
MOVL C01172 V=800.0 PL=0
MOVL C01173 V=800.0 PL=0
MOVL C01174 V=800.0 PL=0
MOVL C01175 V=800.0 PL=0
MOVL C01176 V=800.0 PL=0
MOVL C01177 V=800.0 PL=0
MOVL C01178 V=800.0 PL=0
MOVL C01179 V=800.0 PL=0
MOVL C01180 V=800.0 PL=0
MOVL C01181 V=800.0 PL=0
MOVL C01182 V=800.0 PL=0
MOVL C01183 V=800.0 PL=0
MOVL C01184 V=800.0 PL=0
MOVL C01185 V=800.0 PL=0
MOVL C01186 V=800.0 PL=0
MOVL C01187 V=800.0 PL=0
MOVL C01188 V=800.0 PL=0
MOVL C01189 V=800.0 PL=0
MOVL C01190 V=800.0 PL=0
MOVL C01191 V=800.0 PL=0
MOVL C01192 V=800.0 PL=0
MOVL C01193 V=800.0 PL=0
MOVL C01194 V=800.0 PL=0
MOVL C01195 V=800.0 PL=0
MOVL C01196 V=800.0 PL=0
MOVL C01197 V=800.0 PL=0
MOVL C01198 V=800.0 PL=0
MOVL C01199 V=800.0 PL=0
MOVL C01200 V=800.0 PL=0
MOVL C01201 V=800.0 PL=0
MOVL C01202 V=800.0 PL=0
MOVL C01203 V=800.0 PL=0
MOVL C01204 V=800.0 PL=0
MOVL C01205 V=800.0 PL=0
MOVL C01206 V=800.0 PL=0
MOVL C01207 V=800.0 PL=0
MOVL C01208 V=800.0 PL=0
MOVL C01209 V=800.0 PL=0
MOVL C01210 V=800.0 PL=0
MOVL C01211 V=800.0 PL=0
MOVL C01212 V=800.0 PL=0
MOVL C01213 V=800.0 PL=0
MOVL C01214 V=800.0 PL=0
MOVL C01215 V=800.0 PL=0
MOVL C01216 V=800.0 PL=0
MOVL C01217 V=800.0 PL=0
MOVL C01218 V=800.0 PL=0
MOVL C01219 V=800.0 PL=0
MOVL C01220 V=800.0 PL=0
MOVL C01221 V=800.0 PL=0
MOVL C01222 V=800.0 PL=0
MOVL C01223 V=800.0 PL=0
MOVL C01224 V=800.0 PL=0
MOVL C01225 V=800.0 PL=0
MOVL C01226 V=800.0 PL=0
MOVL C01227 V=800.0 PL=0
MOVL C01228 V=800.0 PL=0
MOVL C01229 V=800.0 PL=0
MOVL C01230 V=800.0 PL=0
MOVL C01231 V=800.0 PL=0
MOVL C01232 V=800.0 PL=0
MOVL C01233 V=800.0 PL=0
MOVL C01234 V=800.0 PL=0
MOVL C01235 V=800.0 PL=0
MOVL C01236 V=800.0 PL=0
MOVL C01237 V=800.0 PL=0
MOVL C01238 V=800.0 PL=0
MOVL C01239 V=800.0 PL=0
MOVL C01240 V=800.0 PL=0
MOVL C01241 V=800.0 PL=0
MOVL C01242 V=800.0 PL=0
MOVL C01243 V=800.0 PL=0
MOVL C01244 V=800.0 PL=0
MOVL C01245 V=800.0 PL=0
MOVL C01246 V=800.0 PL=0
MOVL C01247 V=800.0 PL=0
MOVL C01248 V=800.0 PL=0
MOVL C01249 V=800.0 PL=0
MOVL C01250 V=800.0 PL=0
MOVL C01251 V=800.0 PL=0
MOVL C01252 V=800.0 PL=0
MOVL C01253 V=800.0 PL=0
MOVL C01254 V=800.0 PL=0
MOVL C01255 V=800.0 PL=0
MOVL C01256 V=800.0 PL=0
MOVL C01257 V=800.0 PL=0
MOVL C01258 V=800.0 PL=0
MOVL C01259 V=800.0 PL=0
MOVL C01260 V=800.0 PL=0
MOVL C01261 V=800.0 PL=0
MOVL C01262 V=800.0 PL=0
MOVL C01263 V=800.0 PL=0
MOVL C01264 V=800.0 PL=0
MOVL C01265 V=800.0 PL=0
MOVL C01266 V=800.0 PL=0
MOVL C01267 V=800.0 PL=0
MOVL C01268 V=800.0 PL=0
MOVL C01269 V=800.0 PL=0
MOVL C01270 V=800.0 PL=0
MOVL C01271 V=800.0 PL=0
MOVL C01272 V=800.0 PL=0
MOVL C01273 V=800.0 PL=0
MOVL C01274 V=800.0 PL=0
MOVL C01275 V=800.0 PL=0
MOVL C01276 V=800.0 PL=0
MOVL C01277 V=800.0 PL=0
MOVL C01278 V=800.0 PL=0
MOVL C01279 V=800.0 PL=0
MOVL C01280 V=800.0 PL=0
MOVL C01281 V=800.0 PL=0
MOVL C01282 V=800.0 PL=0
MOVL C01283 V=800.0 PL=0
MOVL C01284 V=800.0 PL=0
MOVL C01285 V=800.0 PL=0
MOVL C01286 V=800.0 PL=0
MOVL C01287 V=800.0 PL=0
MOVL C01288 V=800.0 PL=0
MOVL C01289 V=800.0 PL=0
MOVL C01290 V=800.0 PL=0
MOVL C01291 V=800.0 PL=0
MOVL C01292 V=800.0 PL=0
MOVL C01293 V=800.0 PL=0
MOVL C01294 V=800.0 PL=0
MOVL C01295 V=800.0 PL=0
MOVL C01296 V=800.0 PL=0
MOVL C01297 V=800.0 PL=0
MOVL C01298 V=800.0 PL=0
MOVL C01299 V=800.0 PL=0
MOVL C01300 V=800.0 PL=0
MOVL C01301 V=800.0 PL=0
MOVL C01302 V=800.0 PL=0
MOVL C01303 V=800.0 PL=0
MOVL C01304 V=800.0 PL=0
MOVL C01305 V=800.0 PL=0
MOVL C01306 V=800.0 PL=0
MOVL C01307 V=800.0 PL=0
MOVL C01308 V=800.0 PL=0
MOVL C01309 V=800.0 PL=0
MOVL C01310 V=800.0 PL=0
MOVL C01311 V=800.0 PL=0
MOVL C01312 V=800.0 PL=0
MOVL C01313 V=800.0 PL=0
MOVL C01314 V=800.0 PL=0
MOVL C01315 V=800.0 PL=0
MOVL C01316 V=800.0 PL=0
MOVL C01317 V=800.0 PL=0
MOVL C01318 V=800.0 PL=0
MOVL C01319 V=800.0 PL=0
MOVL C01320 V=800.0 PL=0
MOVL C01321 V=800.0 PL=0
MOVL C01322 V=800.0 PL=0
MOVL C01323 V=800.0 PL=0
MOVL C01324 V=800.0 PL=0
MOVL C01325 V=800.0 PL=0
MOVL C01326 V=800.0 PL=0
MOVL C01327 V=800.0 PL=0
MOVL C01328 V=800.0 PL=0
MOVL C01329 V=800.0 PL=0
MOVL C01330 V=800.0 PL=0
MOVL C01331 V=800.0 PL=0
MOVL C01332 V=800.0 PL=0
MOVL C01333 V=800.0 PL=0
MOVL C01334 V=800.0 PL=0
MOVL C01335 V=800.0 PL=0
MOVL C01336 V=800.0 PL=0
MOVL C01337 V=800.0 PL=0
MOVL C01338 V=800.0 PL=0
MOVL C01339 V=800.0 PL=0
MOVL C01340 V=800.0 PL=0
MOVL C01341 V=800.0 PL=0
MOVL C01342 V=800.0 PL=0
MOVL C01343 V=800.0 PL=0
MOVL C01344 V=800.0 PL=0
MOVL C01345 V=800.0 PL=0
MOVL C01346 V=800.0 PL=0
MOVL C01347 V=800.0 PL=0
MOVL C01348 V=800.0 PL=0
MOVL C01349 V=800.0 PL=0
MOVL C01350 V=800.0 PL=0
MOVL C01351 V=800.0 PL=0
MOVL C01352 V=800.0 PL=0
MOVL C01353 V=800.0 PL=0
MOVL C01354 V=800.0 PL=0
MOVL C01355 V=800.0 PL=0
MOVL C01356 V=800.0 PL=0
MOVL C01357 V=800.0 PL=0
MOVL C01358 V=800.0 PL=0
MOVL C01359 V=800.0 PL=0
MOVL C01360 V=800.0 PL=0
MOVL C01361 V=800.0 PL=0
MOVL C01362 V=800.0 PL=0
MOVL C01363 V=800.0 PL=0
MOVL C01364 V=800.0 PL=0
MOVL C01365 V=800.0 PL=0
MOVL C01366 V=800.0 PL=0
MOVL C01367 V=800.0 PL=0
MOVL C01368 V=800.0 PL=0
MOVL C01369 V=800.0 PL=0
MOVL C01370 V=800.0 PL=0
MOVL C01371 V=800.0 PL=0
MOVL C01372 V=800.0 PL=0
MOVL C01373 V=800.0 PL=0
MOVL C01374 V=800.0 PL=0
MOVL C01375 V=800.0 PL=0
MOVL C01376 V=800.0 PL=0
MOVL C01377 V=800.0 PL=0
MOVL C01378 V=800.0 PL=0
MOVL C01379 V=800.0 PL=0
MOVL C01380 V=800.0 PL=0
MOVL C01381 V=800.0 PL=0
MOVL C01382 V=800.0 PL=0
MOVL C01383 V=800.0 PL=0
MOVL C01384 V=800.0 PL=0
MOVL C01385 V=800.0 PL=0
MOVL C01386 V=800.0 PL=0
MOVL C01387 V=800.0 PL=0
MOVL C01388 V=800.0 PL=0
MOVL C01389 V=800.0 PL=0
MOVL C01390 V=800.0 PL=0
MOVL C01391 V=800.0 PL=0
MOVL C01392 V=800.0 PL=0
MOVL C01393 V=800.0 PL=0
MOVL C01394 V=800.0 PL=0
MOVL C01395 V=800.0 PL=0
MOVL C01396 V=800.0 PL=0
MOVL C01397 V=800.0 PL=0
MOVL C01398 V=800.0 PL=0
MOVL C01399 V=800.0 PL=0
MOVL C01400 V=800.0 PL=0
MOVL C01401 V=800.0 PL=0
MOVL C01402 V=800.0 PL=0
MOVL C01403 V=800.0 PL=0
MOVL C01404 V=800.0 PL=0
MOVL C01405 V=800.0 PL=0
MOVL C01406 V=800.0 PL=0
MOVL C01407 V=800.0 PL=0
MOVL C01408 V=800.0 PL=0
MOVL C01409 V=800.0 PL=0
MOVL C01410 V=800.0 PL=0
MOVL C01411 V=800.0 PL=0
MOVL C01412 V=800.0 PL=0
MOVL C01413 V=800.0 PL=0
MOVL C01414 V=800.0 PL=0
MOVL C01415 V=800.0 PL=0
MOVL C01416 V=800.0 PL=0
MOVL C01417 V=800.0 PL=0
MOVL C01418 V=800.0 PL=0
MOVL C01419 V=800.0 PL=0
MOVL C01420 V=800.0 PL=0
MOVL C01421 V=800.0 PL=0
MOVL C01422 V=800.0 PL=0
MOVL C01423 V=800.0 PL=0
MOVL C01424 V=800.0 PL=0
MOVL C01425 V=800.0 PL=0
MOVL C01426 V=800.0 PL=0
MOVL C01427 V=800.0 PL=0
MOVL C01428 V=800.0 PL=0
MOVL C01429 V=800.0 PL=0
MOVL C01430 V=800.0 PL=0
MOVL C01431 V=800.0 PL=0
MOVL C01432 V=800.0 PL=0
MOVL C01433 V=800.0 PL=0
MOVL C01434 V=800.0 PL=0
MOVL C01435 V=800.0 PL=0
MOVL C01436 V=800.0 PL=0
MOVL C01437 V=800.0 PL=0
MOVL C01438 V=800.0 PL=0
MOVL C01439 V=800.0 PL=0
MOVL C01440 V=800.0 PL=0
MOVL C01441 V=800.0 PL=0
MOVL C01442 V=800.0 PL=0
MOVL C01443 V=800.0 PL=0
MOVL C01444 V=800.0 PL=0
MOVL C01445 V=800.0 PL=0
MOVL C01446 V=800.0 PL=0
MOVL C01447 V=800.0 PL=0
MOVL C01448 V=800.0 PL=0
MOVL C01449 V=800.0 PL=0
MOVL C01450 V=800.0 PL=0
MOVL C01451 V=800.0 PL=0
MOVL C01452 V=800.0 PL=0
MOVL C01453 V=800.0 PL=0
MOVL C01454 V=800.0 PL=0
MOVL C01455 V=800.0 PL=0
MOVL C01456 V=800.0 PL=0
MOVL C01457 V=800.0 PL=0
MOVL C01458 V=800.0 PL=0
MOVL C01459 V=800.0 PL=0
MOVL C01460 V=800.0 PL=0
MOVL C01461 V=800.0 PL=0
MOVL C01462 V=800.0 PL=0
MOVL C01463 V=800.0 PL=0
MOVL C01464 V=800.0 PL=0
MOVL C01465 V=800.0 PL=0
MOVL C01466 V=800.0 PL=0
MOVL C01467 V=800.0 PL=0
MOVL C01468 V=800.0 PL=0
MOVL C01469 V=800.0 PL=0
MOVL C01470 V=800.0 PL=0
MOVL C01471 V=800.0 PL=0
MOVL C01472 V=800.0 PL=0
MOVL C01473 V=800.0 PL=0
MOVL C01474 V=800.0 PL=0
MOVL C01475 V=800.0 PL=0
MOVL C01476 V=800.0 PL=0
MOVL C01477 V=800.0 PL=0
MOVL C01478 V=800.0 PL=0
MOVL C01479 V=800.0 PL=0
MOVL C01480 V=800.0 PL=0
MOVL C01481 V=800.0 PL=0
MOVL C01482 V=800.0 PL=0
MOVL C01483 V=800.0 PL=0
MOVL C01484 V=800.0 PL=0
MOVL C01485 V=800.0 PL=0
MOVL C01486 V=800.0 PL=0
MOVL C01487 V=800.0 PL=0
MOVL C01488 V=800.0 PL=0
MOVL C01489 V=800.0 PL=0
MOVL C01490 V=800.0 PL=0
MOVL C01491 V=800.0 PL=0
MOVL C01492 V=800.0 PL=0
MOVL C01493 V=800.0 PL=0
MOVL C01494 V=800.0 PL=0
MOVL C01495 V=800.0 PL=0
MOVL C01496 V=800.0 PL=0
MOVL C01497 V=800.0 PL=0
MOVL C01498 V=800.0 PL=0
MOVL C01499 V=800.0 PL=0
MOVL C01500 V=800.0 PL=0
MOVL C01501 V=800.0 PL=0
MOVL C01502 V=800.0 PL=0
MOVL C01503 V=800.0 PL=0
MOVL C01504 V=800.0 PL=0
MOVL C01505 V=800.0 PL=0
MOVL C01506 V=800.0 PL=0
MOVL C01507 V=800.0 PL=0
MOVL C01508 V=800.0 PL=0
MOVL C01509 V=800.0 PL=0
MOVL C01510 V=800.0 PL=0
MOVL C01511 V=800.0 PL=0
MOVL C01512 V=800.0 PL=0
MOVL C01513 V=800.0 PL=0
MOVL C01514 V=800.0 PL=0
MOVL C01515 V=800.0 PL=0
MOVL C01516 V=800.0 PL=0
MOVL C01517 V=800.0 PL=0
MOVL C01518 V=800.0 PL=0
MOVL C01519 V=800.0 PL=0
MOVL C01520 V=800.0 PL=0
MOVL C01521 V=800.0 PL=0
MOVL C01522 V=800.0 PL=0
MOVL C01523 V=800.0 PL=0
MOVL C01524 V=800.0 PL=0
MOVL C01525 V=800.0 PL=0
MOVL C01526 V=800.0 PL=0
MOVL C01527 V=800.0 PL=0
MOVL C01528 V=800.0 PL=0
MOVL C01529 V=800.0 PL=0
MOVL C01530 V=800.0 PL=0
MOVL C01531 V=800.0 PL=0
MOVL C01532 V=800.0 PL=0
MOVL C01533 V=800.0 PL=0
MOVL C01534 V=800.0 PL=0
MOVL C01535 V=800.0 PL=0
MOVL C01536 V=800.0 PL=0
MOVL C01537 V=800.0 PL=0
MOVL C01538 V=800.0 PL=0
MOVL C01539 V=800.0 PL=0
MOVL C01540 V=800.0 PL=0
MOVL C01541 V=800.0 PL=0
MOVL C01542 V=800.0 PL=0
MOVL C01543 V=800.0 PL=0
MOVL C01544 V=800.0 PL=0
MOVL C01545 V=800.0 PL=0
MOVL C01546 V=800.0 PL=0
MOVL C01547 V=800.0 PL=0
MOVL C01548 V=800.0 PL=0
MOVL C01549 V=800.0 PL=0
MOVL C01550 V=800.0 PL=0
MOVL C01551 V=800.0 PL=0
MOVL C01552 V=800.0 PL=0
MOVL C01553 V=800.0 PL=0
MOVL C01554 V=800.0 PL=0
MOVL C01555 V=800.0 PL=0
MOVL C01556 V=800.0 PL=0
MOVL C01557 V=800.0 PL=0
MOVL C01558 V=800.0 PL=0
MOVL C01559 V=800.0 PL=0
MOVL C01560 V=800.0 PL=0
MOVL C01561 V=800.0 PL=0
MOVL C01562 V=800.0 PL=0
MOVL C01563 V=800.0 PL=0
MOVL C01564 V=800.0 PL=0
MOVL C01565 V=800.0 PL=0
MOVL C01566 V=800.0 PL=0
MOVL C01567 V=800.0 PL=0
MOVL C01568 V=800.0 PL=0
MOVL C01569 V=800.0 PL=0
MOVL C01570 V=800.0 PL=0
MOVL C01571 V=800.0 PL=0
MOVL C01572 V=800.0 PL=0
MOVL C01573 V=800.0 PL=0
MOVL C01574 V=800.0 PL=0
MOVL C01575 V=800.0 PL=0
MOVL C01576 V=800.0 PL=0
MOVL C01577 V=800.0 PL=0
MOVL C01578 V=800.0 PL=0
MOVL C01579 V=800.0 PL=0
MOVL C01580 V=800.0 PL=0
MOVL C01581 V=800.0 PL=0
MOVL C01582 V=800.0 PL=0
MOVL C01583 V=800.0 PL=0
MOVL C01584 V=800.0 PL=0
MOVL C01585 V=800.0 PL=0
MOVL C01586 V=800.0 PL=0
MOVL C01587 V=800.0 PL=0
MOVL C01588 V=800.0 PL=0
MOVL C01589 V=800.0 PL=0
MOVL C01590 V=800.0 PL=0
MOVL C01591 V=800.0 PL=0
MOVL C01592 V=800.0 PL=0
MOVL C01593 V=800.0 PL=0
MOVL C01594 V=800.0 PL=0
MOVL C01595 V=800.0 PL=0
MOVL C01596 V=800.0 PL=0
MOVL C01597 V=800.0 PL=0
MOVL C01598 V=800.0 PL=0
MOVL C01599 V=800.0 PL=0
MOVL C01600 V=800.0 PL=0
MOVL C01601 V=800.0 PL=0
MOVL C01602 V=800.0 PL=0
MOVL C01603 V=800.0 PL=0
MOVL C01604 V=800.0 PL=0
MOVL C01605 V=800.0 PL=0
MOVL C01606 V=800.0 PL=0
MOVL C01607 V=800.0 PL=0
MOVL C01608 V=800.0 PL=0
MOVL C01609 V=800.0 PL=0
MOVL C01610 V=800.0 PL=0
MOVL C01611 V=800.0 PL=0
MOVL C01612 V=800.0 PL=0
MOVL C01613 V=800.0 PL=0
MOVL C01614 V=800.0 PL=0
MOVL C01615 V=800.0 PL=0
MOVL C01616 V=800.0 PL=0
MOVL C01617 V=800.0 PL=0
MOVL C01618 V=800.0 PL=0
MOVL C01619 V=800.0 PL=0
MOVL C01620 V=800.0 PL=0
MOVL C01621 V=800.0 PL=0
MOVL C01622 V=800.0 PL=0
MOVL C01623 V=800.0 PL=0
MOVL C01624 V=800.0 PL=0
MOVL C01625 V=800.0 PL=0
MOVL C01626 V=800.0 PL=0
MOVL C01627 V=800.0 PL=0
MOVL C01628 V=800.0 PL=0
MOVL C01629 V=800.0 PL=0
MOVL C01630 V=800.0 PL=0
MOVL C01631 V=800.0 PL=0
MOVL C01632 V=800.0 PL=0
MOVL C01633 V=800.0 PL=0
MOVL C01634 V=800.0 PL=0
MOVL C01635 V=800.0 PL=0
MOVL C01636 V=800.0 PL=0
MOVL C01637 V=800.0 PL=0
MOVL C01638 V=800.0 PL=0
MOVL C01639 V=800.0 PL=0
MOVL C01640 V=800.0 PL=0
MOVL C01641 V=800.0 PL=0
MOVL C01642 V=800.0 PL=0
MOVL C01643 V=800.0 PL=0
MOVL C01644 V=800.0 PL=0
MOVL C01645 V=800.0 PL=0
MOVL C01646 V=800.0 PL=0
MOVL C01647 V=800.0 PL=0
MOVL C01648 V=800.0 PL=0
MOVL C01649 V=800.0 PL=0
MOVL C01650 V=800.0 PL=0
MOVL C01651 V=800.0 PL=0
MOVL C01652 V=800.0 PL=0
MOVL C01653 V=800.0 PL=0
MOVL C01654 V=800.0 PL=0
MOVL C01655 V=800.0 PL=0
MOVL C01656 V=800.0 PL=0
MOVL C01657 V=800.0 PL=0
MOVL C01658 V=800.0 PL=0
MOVL C01659 V=800.0 PL=0
MOVL C01660 V=800.0 PL=0
MOVL C01661 V=800.0 PL=0
MOVL C01662 V=800.0 PL=0
MOVL C01663 V=800.0 PL=0
MOVL C01664 V=800.0 PL=0
MOVL C01665 V=800.0 PL=0
MOVL C01666 V=800.0 PL=0
MOVL C01667 V=800.0 PL=0
MOVL C01668 V=800.0 PL=0
MOVL C01669 V=800.0 PL=0
MOVL C01670 V=800.0 PL=0
MOVL C01671 V=800.0 PL=0
MOVL C01672 V=800.0 PL=0
MOVL C01673 V=800.0 PL=0
MOVL C01674 V=800.0 PL=0
MOVL C01675 V=800.0 PL=0
MOVL C01676 V=800.0 PL=0
MOVL C01677 V=800.0 PL=0
MOVL C01678 V=800.0 PL=0
MOVL C01679 V=800.0 PL=0
MOVL C01680 V=800.0 PL=0
MOVL C01681 V=800.0 PL=0
MOVL C01682 V=800.0 PL=0
MOVL C01683 V=800.0 PL=0
MOVL C01684 V=800.0 PL=0
MOVL C01685 V=800.0 PL=0
MOVL C01686 V=800.0 PL=0
MOVL C01687 V=800.0 PL=0
MOVL C01688 V=800.0 PL=0
MOVL C01689 V=800.0 PL=0
MOVL C01690 V=800.0 PL=0
MOVL C01691 V=800.0 PL=0
MOVL C01692 V=800.0 PL=0
MOVL C01693 V=800.0 PL=0
MOVL C01694 V=800.0 PL=0
MOVL C01695 V=800.0 PL=0
MOVL C01696 V=800.0 PL=0
MOVL C01697 V=800.0 PL=0
MOVL C01698 V=800.0 PL=0
MOVL C01699 V=800.0 PL=0
MOVL C01700 V=800.0 PL=0
MOVL C01701 V=800.0 PL=0
MOVL C01702 V=800.0 PL=0
MOVL C01703 V=800.0 PL=0
MOVL C01704 V=800.0 PL=0
MOVL C01705 V=800.0 PL=0
MOVL C01706 V=800.0 PL=0
MOVL C01707 V=800.0 PL=0
MOVL C01708 V=800.0 PL=0
MOVL C01709 V=800.0 PL=0
MOVL C01710 V=800.0 PL=0
MOVL C01711 V=800.0 PL=0
MOVL C01712 V=800.0 PL=0
MOVL C01713 V=800.0 PL=0
MOVL C01714 V=800.0 PL=0
MOVL C01715 V=800.0 PL=0
MOVL C01716 V=800.0 PL=0
MOVL C01717 V=800.0 PL=0
MOVL C01718 V=800.0 PL=0
MOVL C01719 V=800.0 PL=0
MOVL C01720 V=800.0 PL=0
MOVL C01721 V=800.0 PL=0
MOVL C01722 V=800.0 PL=0
MOVL C01723 V=800.0 PL=0
MOVL C01724 V=800.0 PL=0
MOVL C01725 V=800.0 PL=0
MOVL C01726 V=800.0 PL=0
MOVL C01727 V=800.0 PL=0
MOVL C01728 V=800.0 PL=0
MOVL C01729 V=800.0 PL=0
MOVL C01730 V=800.0 PL=0
MOVL C01731 V=800.0 PL=0
MOVL C01732 V=800.0 PL=0
MOVL C01733 V=800.0 PL=0
MOVL C01734 V=800.0 PL=0
MOVL C01735 V=800.0 PL=0
MOVL C01736 V=800.0 PL=0
MOVL C01737 V=800.0 PL=0
MOVL C01738 V=800.0 PL=0
MOVL C01739 V=800.0 PL=0
MOVL C01740 V=800.0 PL=0
MOVL C01741 V=800.0 PL=0
MOVL C01742 V=800.0 PL=0
MOVL C01743 V=800.0 PL=0
MOVL C01744 V=800.0 PL=0
MOVL C01745 V=800.0 PL=0
MOVL C01746 V=800.0 PL=0
MOVL C01747 V=800.0 PL=0
MOVL C01748 V=800.0 PL=0
MOVL C01749 V=800.0 PL=0
MOVL C01750 V=800.0 PL=0
MOVL C01751 V=800.0 PL=0
MOVL C01752 V=800.0 PL=0
MOVL C01753 V=800.0 PL=0
MOVL C01754 V=800.0 PL=0
MOVL C01755 V=800.0 PL=0
MOVL C01756 V=800.0 PL=0
MOVL C01757 V=800.0 PL=0
MOVL C01758 V=800.0 PL=0
MOVL C01759 V=800.0 PL=0
MOVL C01760 V=800.0 PL=0
MOVL C01761 V=800.0 PL=0
MOVL C01762 V=800.0 PL=0
MOVL C01763 V=800.0 PL=0
MOVL C01764 V=800.0 PL=0
MOVL C01765 V=800.0 PL=0
MOVL C01766 V=800.0 PL=0
MOVL C01767 V=800.0 PL=0
MOVL C01768 V=800.0 PL=0
MOVL C01769 V=800.0 PL=0
MOVL C01770 V=800.0 PL=0
MOVL C01771 V=800.0 PL=0
MOVL C01772 V=800.0 PL=0
MOVL C01773 V=800.0 PL=0
MOVL C01774 V=800.0 PL=0
MOVL C01775 V=800.0 PL=0
MOVL C01776 V=800.0 PL=0
MOVL C01777 V=800.0 PL=0
MOVL C01778 V=800.0 PL=0
MOVL C01779 V=800.0 PL=0
MOVL C01780 V=800.0 PL=0
MOVL C01781 V=800.0 PL=0
MOVL C01782 V=800.0 PL=0
MOVL C01783 V=800.0 PL=0
MOVL C01784 V=800.0 PL=0
MOVL C01785 V=800.0 PL=0
MOVL C01786 V=800.0 PL=0
MOVL C01787 V=800.0 PL=0
MOVL C01788 V=800.0 PL=0
MOVL C01789 V=800.0 PL=0
MOVL C01790 V=800.0 PL=0
MOVL C01791 V=800.0 PL=0
MOVL C01792 V=800.0 PL=0
MOVL C01793 V=800.0 PL=0
MOVL C01794 V=800.0 PL=0
MOVL C01795 V=800.0 PL=0
MOVL C01796 V=800.0 PL=0
MOVL C01797 V=800.0 PL=0
MOVL C01798 V=800.0 PL=0
MOVL C01799 V=800.0 PL=0
MOVL C01800 V=800.0 PL=0
MOVL C01801 V=800.0 PL=0
MOVL C01802 V=800.0 PL=0
MOVL C01803 V=800.0 PL=0
MOVL C01804 V=800.0 PL=0
MOVL C01805 V=800.0 PL=0
MOVL C01806 V=800.0 PL=0
MOVL C01807 V=800.0 PL=0
MOVL C01808 V=800.0 PL=0
MOVL C01809 V=800.0 PL=0
MOVL C01810 V=800.0 PL=0
MOVL C01811 V=800.0 PL=0
MOVL C01812 V=800.0 PL=0
MOVL C01813 V=800.0 PL=0
MOVL C01814 V=800.0 PL=0
MOVL C01815 V=800.0 PL=0
MOVL C01816 V=800.0 PL=0
MOVL C01817 V=800.0 PL=0
MOVL C01818 V=800.0 PL=0
MOVL C01819 V=800.0 PL=0
MOVL C01820 V=800.0 PL=0
MOVL C01821 V=800.0 PL=0
MOVL C01822 V=800.0 PL=0
MOVL C01823 V=800.0 PL=0
MOVL C01824 V=800.0 PL=0
MOVL C01825 V=800.0 PL=0
MOVL C01826 V=800.0 PL=0
MOVL C01827 V=800.0 PL=0
MOVL C01828 V=800.0 PL=0
MOVL C01829 V=800.0 PL=0
MOVL C01830 V=800.0 PL=0
MOVL C01831 V=800.0 PL=0
MOVL C01832 V=800.0 PL=0
MOVL C01833 V=800.0 PL=0
MOVL C01834 V=800.0 PL=0
MOVL C01835 V=800.0 PL=0
MOVL C01836 V=800.0 PL=0
MOVL C01837 V=800.0 PL=0
MOVL C01838 V=800.0 PL=0
MOVL C01839 V=800.0 PL=0
MOVL C01840 V=800.0 PL=0
MOVL C01841 V=800.0 PL=0
MOVL C01842 V=800.0 PL=0
MOVL C01843 V=800.0 PL=0
MOVL C01844 V=800.0 PL=0
MOVL C01845 V=800.0 PL=0
MOVL C01846 V=800.0 PL=0
MOVL C01847 V=800.0 PL=0
MOVL C01848 V=800.0 PL=0
MOVL C01849 V=800.0 PL=0
MOVL C01850 V=800.0 PL=0
MOVL C01851 V=800.0 PL=0
MOVL C01852 V=800.0 PL=0
MOVL C01853 V=800.0 PL=0
MOVL C01854 V=800.0 PL=0
MOVL C01855 V=800.0 PL=0
MOVL C01856 V=800.0 PL=0
MOVL C01857 V=800.0 PL=0
MOVL C01858 V=800.0 PL=0
MOVL C01859 V=800.0 PL=0
MOVL C01860 V=800.0 PL=0
MOVL C01861 V=800.0 PL=0
MOVL C01862 V=800.0 PL=0
MOVL C01863 V=800.0 PL=0
MOVL C01864 V=800.0 PL=0
MOVL C01865 V=800.0 PL=0
MOVL C01866 V=800.0 PL=0
MOVL C01867 V=800.0 PL=0
MOVL C01868 V=800.0 PL=0
MOVL C01869 V=800.0 PL=0
MOVL C01870 V=800.0 PL=0
MOVL C01871 V=800.0 PL=0
MOVL C01872 V=800.0 PL=0
MOVL C01873 V=800.0 PL=0
MOVL C01874 V=800.0 PL=0
MOVL C01875 V=800.0 PL=0
MOVL C01876 V=800.0 PL=0
MOVL C01877 V=800.0 PL=0
MOVL C01878 V=800.0 PL=0
MOVL C01879 V=800.0 PL=0
MOVL C01880 V=800.0 PL=0
MOVL C01881 V=800.0 PL=0
MOVL C01882 V=800.0 PL=0
MOVL C01883 V=800.0 PL=0
MOVL C01884 V=800.0 PL=0
MOVL C01885 V=800.0 PL=0
MOVL C01886 V=800.0 PL=0
MOVL C01887 V=800.0 PL=0
MOVL C01888 V=800.0 PL=0
MOVL C01889 V=800.0 PL=0
MOVL C01890 V=800.0 PL=0
MOVL C01891 V=800.0 PL=0
MOVL C01892 V=800.0 PL=0
MOVL C01893 V=800.0 PL=0
MOVL C01894 V=800.0 PL=0
MOVL C01895 V=800.0 PL=0
MOVL C01896 V=800.0 PL=0
MOVL C01897 V=800.0 PL=0
MOVL C01898 V=800.0 PL=0
MOVL C01899 V=800.0 PL=0
MOVL C01900 V=800.0 PL=0
MOVL C01901 V=800.0 PL=0
MOVL C01902 V=800.0 PL=0
MOVL C01903 V=800.0 PL=0
MOVL C01904 V=800.0 PL=0
MOVL C01905 V=800.0 PL=0
MOVL C01906 V=800.0 PL=0
MOVL C01907 V=800.0 PL=0
MOVL C01908 V=800.0 PL=0
MOVL C01909 V=800.0 PL=0
MOVL C01910 V=800.0 PL=0
MOVL C01911 V=800.0 PL=0
MOVL C01912 V=800.0 PL=0
MOVL C01913 V=800.0 PL=0
MOVL C01914 V=800.0 PL=0
MOVL C01915 V=800.0 PL=0
MOVL C01916 V=800.0 PL=0
MOVL C01917 V=800.0 PL=0
MOVL C01918 V=800.0 PL=0
MOVL C01919 V=800.0 PL=0
MOVL C01920 V=800.0 PL=0
MOVL C01921 V=800.0 PL=0
MOVL C01922 V=800.0 PL=0
MOVL C01923 V=800.0 PL=0
MOVL C01924 V=800.0 PL=0
MOVL C01925 V=800.0 PL=0
MOVL C01926 V=800.0 PL=0
MOVL C01927 V=800.0 PL=0
MOVL C01928 V=800.0 PL=0
MOVL C01929 V=800.0 PL=0
MOVL C01930 V=800.0 PL=0
MOVL C01931 V=800.0 PL=0
MOVL C01932 V=800.0 PL=0
MOVL C01933 V=800.0 PL=0
MOVL C01934 V=800.0 PL=0
MOVL C01935 V=800.0 PL=0
MOVL C01936 V=800.0 PL=0
MOVL C01937 V=800.0 PL=0
MOVL C01938 V=800.0 PL=0
MOVL C01939 V=800.0 PL=0
MOVL C01940 V=800.0 PL=0
MOVL C01941 V=800.0 PL=0
MOVL C01942 V=800.0 PL=0
MOVL C01943 V=800.0 PL=0
MOVL C01944 V=800.0 PL=0
MOVL C01945 V=800.0 PL=0
MOVL C01946 V=800.0 PL=0
MOVL C01947 V=800.0 PL=0
MOVL C01948 V=800.0 PL=0
MOVL C01949 V=800.0 PL=0
MOVL C01950 V=800.0 PL=0
MOVL C01951 V=800.0 PL=0
MOVL C01952 V=800.0 PL=0
MOVL C01953 V=800.0 PL=0
MOVL C01954 V=800.0 PL=0
MOVL C01955 V=800.0 PL=0
MOVL C01956 V=800.0 PL=0
MOVL C01957 V=800.0 PL=0
MOVL C01958 V=800.0 PL=0
MOVL C01959 V=800.0 PL=0
MOVL C01960 V=800.0 PL=0
MOVL C01961 V=800.0 PL=0
MOVL C01962 V=800.0 PL=0
MOVL C01963 V=800.0 PL=0
MOVL C01964 V=800.0 PL=0
MOVL C01965 V=800.0 PL=0
MOVL C01966 V=800.0 PL=0
MOVL C01967 V=800.0 PL=0
MOVL C01968 V=800.0 PL=0
MOVL C01969 V=800.0 PL=0
MOVL C01970 V=800.0 PL=0
MOVL C01971 V=800.0 PL=0
MOVL C01972 V=800.0 PL=0
MOVL C01973 V=800.0 PL=0
MOVL C01974 V=800.0 PL=0
MOVL C01975 V=800.0 PL=0
MOVL C01976 V=800.0 PL=0
MOVL C01977 V=800.0 PL=0
MOVL C01978 V=800.0 PL=0
MOVL C01979 V=800.0 PL=0
MOVL C01980 V=800.0 PL=0
MOVL C01981 V=800.0 PL=0
MOVL C01982 V=800.0 PL=0
MOVL C01983 V=800.0 PL=0
MOVL C01984 V=800.0 PL=0
MOVL C01985 V=800.0 PL=0
MOVL C01986 V=800.0 PL=0
MOVL C01987 V=800.0 PL=0
MOVL C01988 V=800.0 PL=0
MOVL C01989 V=800.0 PL=0
MOVL C01990 V=800.0 PL=0
MOVL C01991 V=800.0 PL=0
MOVL C01992 V=800.0 PL=0
MOVL C01993 V=800.0 PL=0
MOVL C01994 V=800.0 PL=0
MOVL C01995 V=800.0 PL=0
MOVL C01996 V=800.0 PL=0
MOVL C01997 V=800.0 PL=0
MOVL C01998 V=800.0 PL=0
MOVL C01999 V=800.0 PL=0
MOVL C02000 V=800.0 PL=0
MOVL C02001 V=800.0 PL=0
MOVL C02002 V=800.0 PL=0
MOVL C02003 V=800.0 PL=0
MOVL C02004 V=800.0 PL=0
MOVL C02005 V=800.0 PL=0
MOVL C02006 V=800.0 PL=0
MOVL C02007 V=800.0 PL=0
MOVL C02008 V=800.0 PL=0
MOVL C02009 V=800.0 PL=0
MOVL C02010 V=800.0 PL=0
MOVL C02011 V=800.0 PL=0
MOVL C02012 V=800.0 PL=0
MOVL C02013 V=800.0 PL=0
MOVL C02014 V=800.0 PL=0
MOVL C02015 V=800.0 PL=0
MOVL C02016 V=800.0 PL=0
MOVL C02017 V=800.0 PL=0
MOVL C02018 V=800.0 PL=0
MOVL C02019 V=800.0 PL=0
MOVL C02020 V=800.0 PL=0
MOVL C02021 V=800.0 PL=0
MOVL C02022 V=800.0 PL=0
MOVL C02023 V=800.0 PL=0
MOVL C02024 V=800.0 PL=0
MOVL C02025 V=800.0 PL=0
MOVL C02026 V=800.0 PL=0
MOVL C02027 V=800.0 PL=0
MOVL C02028 V=800.0 PL=0
MOVL C02029 V=800.0 PL=0
MOVL C02030 V=800.0 PL=0
MOVL C02031 V=800.0 PL=0
MOVL C02032 V=800.0 PL=0
MOVL C02033 V=800.0 PL=0
MOVL C02034 V=800.0 PL=0
MOVL C02035 V=800.0 PL=0
MOVL C02036 V=800.0 PL=0
MOVL C02037 V=800.0 PL=0
MOVL C02038 V=800.0 PL=0
MOVL C02039 V=800.0 PL=0
MOVL C02040 V=800.0 PL=0
MOVL C02041 V=800.0 PL=0
MOVL C02042 V=800.0 PL=0
MOVL C02043 V=800.0 PL=0
MOVL C02044 V=800.0 PL=0
MOVL C02045 V=800.0 PL=0
MOVL C02046 V=800.0 PL=0
MOVL C02047 V=800.0 PL=0
MOVL C02048 V=800.0 PL=0
MOVL C02049 V=800.0 PL=0
MOVL C02050 V=800.0 PL=0
MOVL C02051 V=800.0 PL=0
MOVL C02052 V=800.0 PL=0
MOVL C02053 V=800.0 PL=0
MOVL C02054 V=800.0 PL=0
MOVL C02055 V=800.0 PL=0
MOVL C02056 V=800.0 PL=0
MOVL C02057 V=800.0 PL=0
MOVL C02058 V=800.0 PL=0
MOVL C02059 V=800.0 PL=0
MOVL C02060 V=800.0 PL=0
MOVL C02061 V=800.0 PL=0
MOVL C02062 V=800.0 PL=0
MOVL C02063 V=800.0 PL=0
MOVL C02064 V=800.0 PL=0
MOVL C02065 V=800.0 PL=0
MOVL C02066 V=800.0 PL=0
MOVL C02067 V=800.0 PL=0
MOVL C02068 V=800.0 PL=0
MOVL C02069 V=800.0 PL=0
MOVL C02070 V=800.0 PL=0
MOVL C02071 V=800.0 PL=0
MOVL C02072 V=800.0 PL=0
MOVL C02073 V=800.0 PL=0
MOVL C02074 V=800.0 PL=0
MOVL C02075 V=800.0 PL=0
MOVL C02076 V=800.0 PL=0
MOVL C02077 V=800.0 PL=0
MOVL C02078 V=800.0 PL=0
MOVL C02079 V=800.0 PL=0
MOVL C02080 V=800.0 PL=0
MOVL C02081 V=800.0 PL=0
MOVL C02082 V=800.0 PL=0
MOVL C02083 V=800.0 PL=0
MOVL C02084 V=800.0 PL=0
MOVL C02085 V=800.0 PL=0
MOVL C02086 V=800.0 PL=0
MOVL C02087 V=800.0 PL=0
MOVL C02088 V=800.0 PL=0
MOVL C02089 V=800.0 PL=0
MOVL C02090 V=800.0 PL=0
MOVL C02091 V=800.0 PL=0
MOVL C02092 V=800.0 PL=0
MOVL C02093 V=800.0 PL=0
MOVL C02094 V=800.0 PL=0
MOVL C02095 V=800.0 PL=0
MOVL C02096 V=800.0 PL=0
MOVL C02097 V=800.0 PL=0
MOVL C02098 V=800.0 PL=0
MOVL C02099 V=800.0 PL=0
MOVL C02100 V=800.0 PL=0
MOVL C02101 V=800.0 PL=0
MOVL C02102 V=800.0 PL=0
MOVL C02103 V=800.0 PL=0
MOVL C02104 V=800.0 PL=0
MOVL C02105 V=800.0 PL=0
MOVL C02106 V=800.0 PL=0
MOVL C02107 V=800.0 PL=0
MOVL C02108 V=800.0 PL=0
MOVL C02109 V=800.0 PL=0
MOVL C02110 V=800.0 PL=0
MOVL C02111 V=800.0 PL=0
MOVL C02112 V=800.0 PL=0
MOVL C02113 V=800.0 PL=0
MOVL C02114 V=800.0 PL=0
MOVL C02115 V=800.0 PL=0
MOVL C02116 V=800.0 PL=0
MOVL C02117 V=800.0 PL=0
MOVL C02118 V=800.0 PL=0
MOVL C02119 V=800.0 PL=0
MOVL C02120 V=800.0 PL=0
MOVL C02121 V=800.0 PL=0
MOVL C02122 V=800.0 PL=0
MOVL C02123 V=800.0 PL=0
MOVL C02124 V=800.0 PL=0
MOVL C02125 V=800.0 PL=0
MOVL C02126 V=800.0 PL=0
MOVL C02127 V=800.0 PL=0
MOVL C02128 V=800.0 PL=0
MOVL C02129 V=800.0 PL=0
MOVL C02130 V=800.0 PL=0
MOVL C02131 V=800.0 PL=0
MOVL C02132 V=800.0 PL=0
MOVL C02133 V=800.0 PL=0
MOVL C02134 V=800.0 PL=0
MOVL C02135 V=800.0 PL=0
MOVL C02136 V=800.0 PL=0
MOVL C02137 V=800.0 PL=0
MOVL C02138 V=800.0 PL=0
MOVL C02139 V=800.0 PL=0
MOVL C02140 V=800.0 PL=0
MOVL C02141 V=800.0 PL=0
MOVL C02142 V=800.0 PL=0
MOVL C02143 V=800.0 PL=0
MOVL C02144 V=800.0 PL=0
MOVL C02145 V=800.0 PL=0
MOVL C02146 V=800.0 PL=0
MOVL C02147 V=800.0 PL=0
MOVL C02148 V=800.0 PL=0
MOVL C02149 V=800.0 PL=0
MOVL C02150 V=800.0 PL=0
MOVL C02151 V=800.0 PL=0
MOVL C02152 V=800.0 PL=0
MOVL C02153 V=800.0 PL=0
MOVL C02154 V=800.0 PL=0
MOVL C02155 V=800.0 PL=0
MOVL C02156 V=800.0 PL=0
MOVL C02157 V=800.0 PL=0
MOVL C02158 V=800.0 PL=0
MOVL C02159 V=800.0 PL=0
MOVL C02160 V=800.0 PL=0
MOVL C02161 V=800.0 PL=0
MOVL C02162 V=800.0 PL=0
MOVL C02163 V=800.0 PL=0
MOVL C02164 V=800.0 PL=0
MOVL C02165 V=800.0 PL=0
MOVL C02166 V=800.0 PL=0
MOVL C02167 V=800.0 PL=0
MOVL C02168 V=800.0 PL=0
